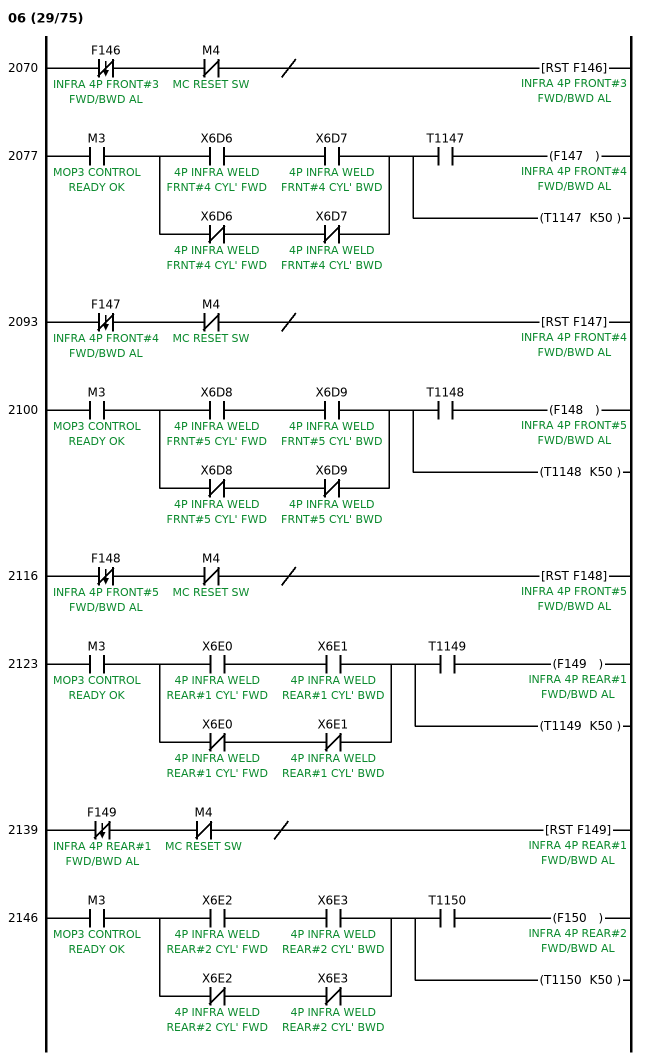
2070  LDFI    F146  ; INFRA 4P FRONT#3 FWD/BWD AL
      ANI     M4  ; MC RESET SW
      INV
      RST     F146  ; INFRA 4P FRONT#3 FWD/BWD AL
2077  LD      M3  ; MOP3 CONTROL READY OK
      LD      X6D6  ; 4P INFRA WELD FRNT#4 CYL' FWD
      AND     X6D7  ; 4P INFRA WELD FRNT#4 CYL' BWD
      LDI     X6D6  ; 4P INFRA WELD FRNT#4 CYL' FWD
      ANI     X6D7  ; 4P INFRA WELD FRNT#4 CYL' BWD
      ORB
      ANB
      MPS
      AND     T1147
      OUT     F147  ; INFRA 4P FRONT#4 FWD/BWD AL
      MPP
      OUT     T1147 K50
2093  LDFI    F147  ; INFRA 4P FRONT#4 FWD/BWD AL
      ANI     M4  ; MC RESET SW
      INV
      RST     F147  ; INFRA 4P FRONT#4 FWD/BWD AL
2100  LD      M3  ; MOP3 CONTROL READY OK
      LD      X6D8  ; 4P INFRA WELD FRNT#5 CYL' FWD
      AND     X6D9  ; 4P INFRA WELD FRNT#5 CYL' BWD
      LDI     X6D8  ; 4P INFRA WELD FRNT#5 CYL' FWD
      ANI     X6D9  ; 4P INFRA WELD FRNT#5 CYL' BWD
      ORB
      ANB
      MPS
      AND     T1148
      OUT     F148  ; INFRA 4P FRONT#5 FWD/BWD AL
      MPP
      OUT     T1148 K50
2116  LDFI    F148  ; INFRA 4P FRONT#5 FWD/BWD AL
      ANI     M4  ; MC RESET SW
      INV
      RST     F148  ; INFRA 4P FRONT#5 FWD/BWD AL
2123  LD      M3  ; MOP3 CONTROL READY OK
      LD      X6E0  ; 4P INFRA WELD REAR#1 CYL' FWD
      AND     X6E1  ; 4P INFRA WELD REAR#1 CYL' BWD
      LDI     X6E0  ; 4P INFRA WELD REAR#1 CYL' FWD
      ANI     X6E1  ; 4P INFRA WELD REAR#1 CYL' BWD
      ORB
      ANB
      MPS
      AND     T1149
      OUT     F149  ; INFRA 4P REAR#1 FWD/BWD AL
      MPP
      OUT     T1149 K50
2139  LDFI    F149  ; INFRA 4P REAR#1 FWD/BWD AL
      ANI     M4  ; MC RESET SW
      INV
      RST     F149  ; INFRA 4P REAR#1 FWD/BWD AL
2146  LD      M3  ; MOP3 CONTROL READY OK
      LD      X6E2  ; 4P INFRA WELD REAR#2 CYL' FWD
      AND     X6E3  ; 4P INFRA WELD REAR#2 CYL' BWD
      LDI     X6E2  ; 4P INFRA WELD REAR#2 CYL' FWD
      ANI     X6E3  ; 4P INFRA WELD REAR#2 CYL' BWD
      ORB
      ANB
      MPS
      AND     T1150
      OUT     F150  ; INFRA 4P REAR#2 FWD/BWD AL
      MPP
      OUT     T1150 K50
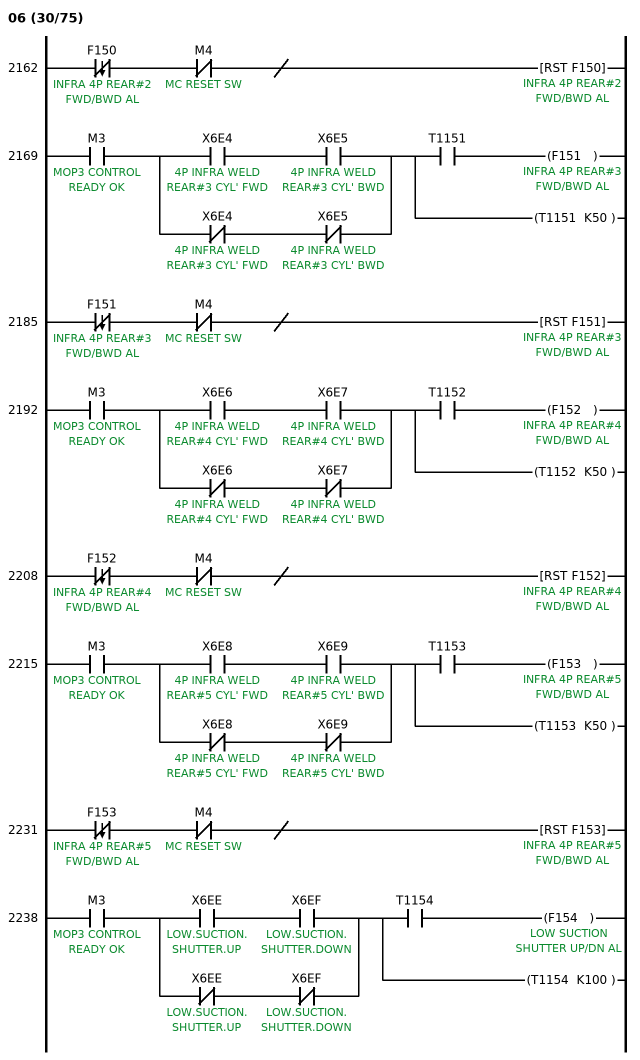
2162  LDFI    F150  ; INFRA 4P REAR#2 FWD/BWD AL
      ANI     M4  ; MC RESET SW
      INV
      RST     F150  ; INFRA 4P REAR#2 FWD/BWD AL
2169  LD      M3  ; MOP3 CONTROL READY OK
      LD      X6E4  ; 4P INFRA WELD REAR#3 CYL' FWD
      AND     X6E5  ; 4P INFRA WELD REAR#3 CYL' BWD
      LDI     X6E4  ; 4P INFRA WELD REAR#3 CYL' FWD
      ANI     X6E5  ; 4P INFRA WELD REAR#3 CYL' BWD
      ORB
      ANB
      MPS
      AND     T1151
      OUT     F151  ; INFRA 4P REAR#3 FWD/BWD AL
      MPP
      OUT     T1151 K50
2185  LDFI    F151  ; INFRA 4P REAR#3 FWD/BWD AL
      ANI     M4  ; MC RESET SW
      INV
      RST     F151  ; INFRA 4P REAR#3 FWD/BWD AL
2192  LD      M3  ; MOP3 CONTROL READY OK
      LD      X6E6  ; 4P INFRA WELD REAR#4 CYL' FWD
      AND     X6E7  ; 4P INFRA WELD REAR#4 CYL' BWD
      LDI     X6E6  ; 4P INFRA WELD REAR#4 CYL' FWD
      ANI     X6E7  ; 4P INFRA WELD REAR#4 CYL' BWD
      ORB
      ANB
      MPS
      AND     T1152
      OUT     F152  ; INFRA 4P REAR#4 FWD/BWD AL
      MPP
      OUT     T1152 K50
2208  LDFI    F152  ; INFRA 4P REAR#4 FWD/BWD AL
      ANI     M4  ; MC RESET SW
      INV
      RST     F152  ; INFRA 4P REAR#4 FWD/BWD AL
2215  LD      M3  ; MOP3 CONTROL READY OK
      LD      X6E8  ; 4P INFRA WELD REAR#5 CYL' FWD
      AND     X6E9  ; 4P INFRA WELD REAR#5 CYL' BWD
      LDI     X6E8  ; 4P INFRA WELD REAR#5 CYL' FWD
      ANI     X6E9  ; 4P INFRA WELD REAR#5 CYL' BWD
      ORB
      ANB
      MPS
      AND     T1153
      OUT     F153  ; INFRA 4P REAR#5 FWD/BWD AL
      MPP
      OUT     T1153 K50
2231  LDFI    F153  ; INFRA 4P REAR#5 FWD/BWD AL
      ANI     M4  ; MC RESET SW
      INV
      RST     F153  ; INFRA 4P REAR#5 FWD/BWD AL
2238  LD      M3  ; MOP3 CONTROL READY OK
      LD      X6EE  ; LOW.SUCTION.SHUTTER.UP
      AND     X6EF  ; LOW.SUCTION.SHUTTER.DOWN
      LDI     X6EE  ; LOW.SUCTION.SHUTTER.UP
      ANI     X6EF  ; LOW.SUCTION.SHUTTER.DOWN
      ORB
      ANB
      MPS
      AND     T1154
      OUT     F154  ; LOW SUCTION SHUTTER UP/DN AL
      MPP
      OUT     T1154 K100
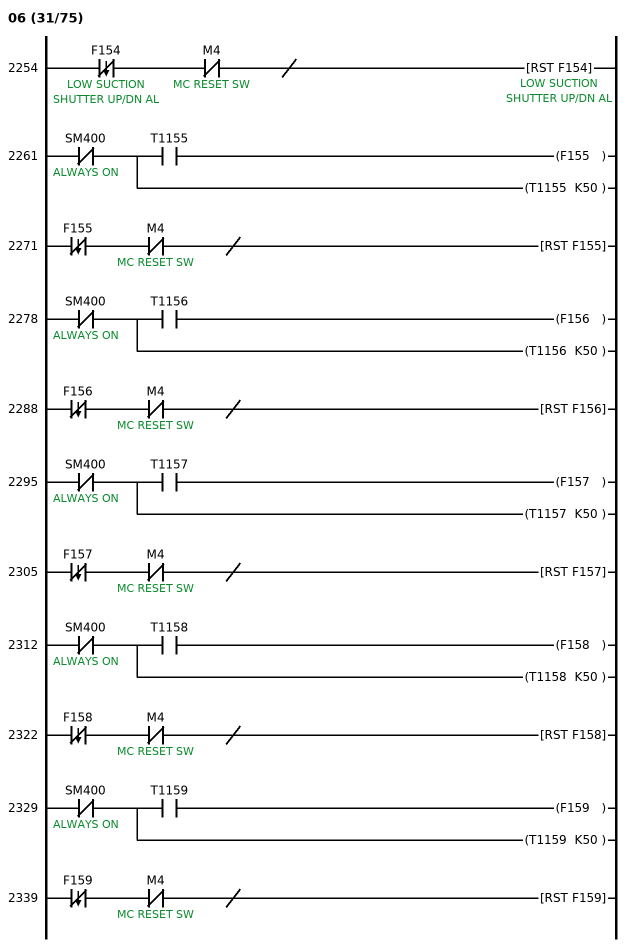
2254  LDFI    F154  ; LOW SUCTION SHUTTER UP/DN AL
      ANI     M4  ; MC RESET SW
      INV
      RST     F154  ; LOW SUCTION SHUTTER UP/DN AL
2261  LDI     SM400  ; ALWAYS ON
      MPS
      AND     T1155
      OUT     F155
      MPP
      OUT     T1155 K50
2271  LDFI    F155
      ANI     M4  ; MC RESET SW
      INV
      RST     F155
2278  LDI     SM400  ; ALWAYS ON
      MPS
      AND     T1156
      OUT     F156
      MPP
      OUT     T1156 K50
2288  LDFI    F156
      ANI     M4  ; MC RESET SW
      INV
      RST     F156
2295  LDI     SM400  ; ALWAYS ON
      MPS
      AND     T1157
      OUT     F157
      MPP
      OUT     T1157 K50
2305  LDFI    F157
      ANI     M4  ; MC RESET SW
      INV
      RST     F157
2312  LDI     SM400  ; ALWAYS ON
      MPS
      AND     T1158
      OUT     F158
      MPP
      OUT     T1158 K50
2322  LDFI    F158
      ANI     M4  ; MC RESET SW
      INV
      RST     F158
2329  LDI     SM400  ; ALWAYS ON
      MPS
      AND     T1159
      OUT     F159
      MPP
      OUT     T1159 K50
2339  LDFI    F159
      ANI     M4  ; MC RESET SW
      INV
      RST     F159
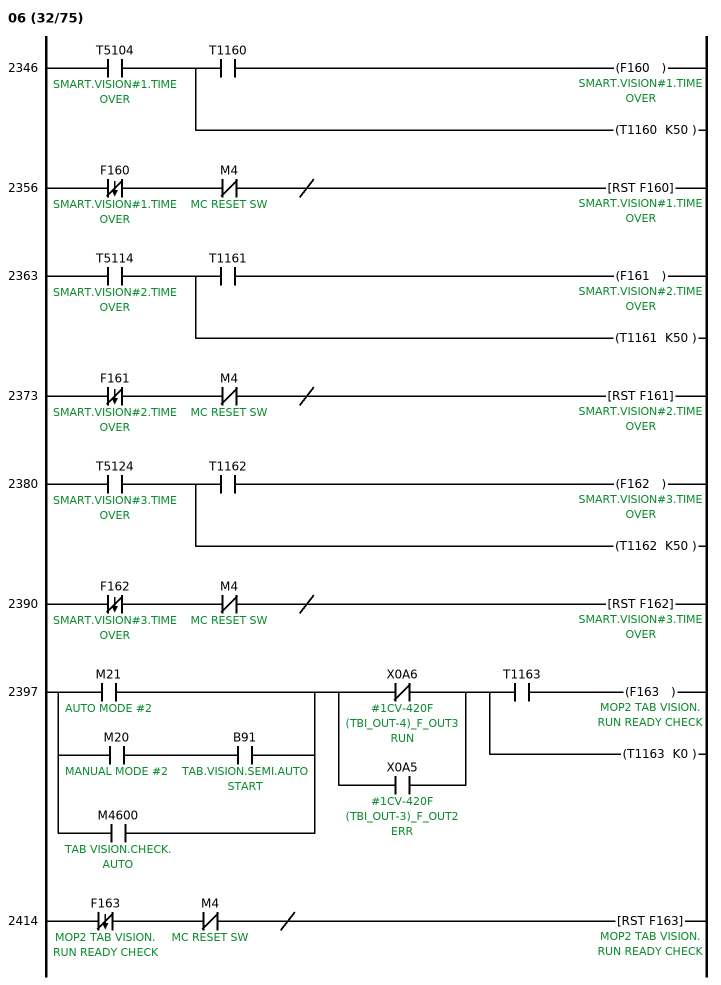
2346  LD      T5104  ; SMART.VISION#1.TIME OVER
      MPS
      AND     T1160
      OUT     F160  ; SMART.VISION#1.TIME OVER
      MPP
      OUT     T1160 K50
2356  LDFI    F160  ; SMART.VISION#1.TIME OVER
      ANI     M4  ; MC RESET SW
      INV
      RST     F160  ; SMART.VISION#1.TIME OVER
2363  LD      T5114  ; SMART.VISION#2.TIME OVER
      MPS
      AND     T1161
      OUT     F161  ; SMART.VISION#2.TIME OVER
      MPP
      OUT     T1161 K50
2373  LDFI    F161  ; SMART.VISION#2.TIME OVER
      ANI     M4  ; MC RESET SW
      INV
      RST     F161  ; SMART.VISION#2.TIME OVER
2380  LD      T5124  ; SMART.VISION#3.TIME OVER
      MPS
      AND     T1162
      OUT     F162  ; SMART.VISION#3.TIME OVER
      MPP
      OUT     T1162 K50
2390  LDFI    F162  ; SMART.VISION#3.TIME OVER
      ANI     M4  ; MC RESET SW
      INV
      RST     F162  ; SMART.VISION#3.TIME OVER
2397  LD      M21  ; AUTO MODE #2
      LD      M20  ; MANUAL MODE #2
      AND     B91  ; TAB.VISION.SEMI.AUTO START
      ORB
      OR      M4600  ; TAB VISION.CHECK.AUTO
      LDI     X0A6  ; #1CV-420F (TBI_OUT-4)_F_OUT3 RUN
      OR      X0A5  ; #1CV-420F (TBI_OUT-3)_F_OUT2 ERR
      ANB
      MPS
      AND     T1163
      OUT     F163  ; MOP2 TAB VISION. RUN READY CHECK
      MPP
      OUT     T1163 K0
2414  LDFI    F163  ; MOP2 TAB VISION. RUN READY CHECK
      ANI     M4  ; MC RESET SW
      INV
      RST     F163  ; MOP2 TAB VISION. RUN READY CHECK
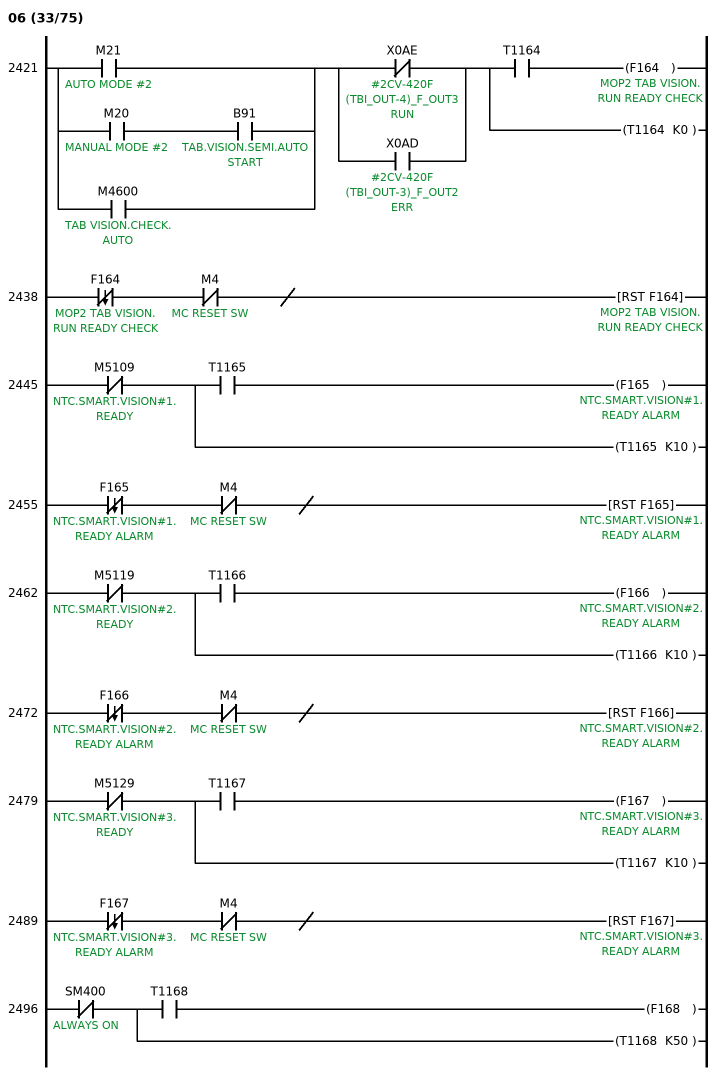
2421  LD      M21  ; AUTO MODE #2
      LD      M20  ; MANUAL MODE #2
      AND     B91  ; TAB.VISION.SEMI.AUTO START
      ORB
      OR      M4600  ; TAB VISION.CHECK.AUTO
      LDI     X0AE  ; #2CV-420F (TBI_OUT-4)_F_OUT3 RUN
      OR      X0AD  ; #2CV-420F (TBI_OUT-3)_F_OUT2 ERR
      ANB
      MPS
      AND     T1164
      OUT     F164  ; MOP2 TAB VISION. RUN READY CHECK
      MPP
      OUT     T1164 K0
2438  LDFI    F164  ; MOP2 TAB VISION. RUN READY CHECK
      ANI     M4  ; MC RESET SW
      INV
      RST     F164  ; MOP2 TAB VISION. RUN READY CHECK
2445  LDI     M5109  ; NTC.SMART.VISION#1.READY
      MPS
      AND     T1165
      OUT     F165  ; NTC.SMART.VISION#1.READY ALARM
      MPP
      OUT     T1165 K10
2455  LDFI    F165  ; NTC.SMART.VISION#1.READY ALARM
      ANI     M4  ; MC RESET SW
      INV
      RST     F165  ; NTC.SMART.VISION#1.READY ALARM
2462  LDI     M5119  ; NTC.SMART.VISION#2.READY
      MPS
      AND     T1166
      OUT     F166  ; NTC.SMART.VISION#2.READY ALARM
      MPP
      OUT     T1166 K10
2472  LDFI    F166  ; NTC.SMART.VISION#2.READY ALARM
      ANI     M4  ; MC RESET SW
      INV
      RST     F166  ; NTC.SMART.VISION#2.READY ALARM
2479  LDI     M5129  ; NTC.SMART.VISION#3.READY
      MPS
      AND     T1167
      OUT     F167  ; NTC.SMART.VISION#3.READY ALARM
      MPP
      OUT     T1167 K10
2489  LDFI    F167  ; NTC.SMART.VISION#3.READY ALARM
      ANI     M4  ; MC RESET SW
      INV
      RST     F167  ; NTC.SMART.VISION#3.READY ALARM
2496  LDI     SM400  ; ALWAYS ON
      MPS
      AND     T1168
      OUT     F168
      MPP
      OUT     T1168 K50
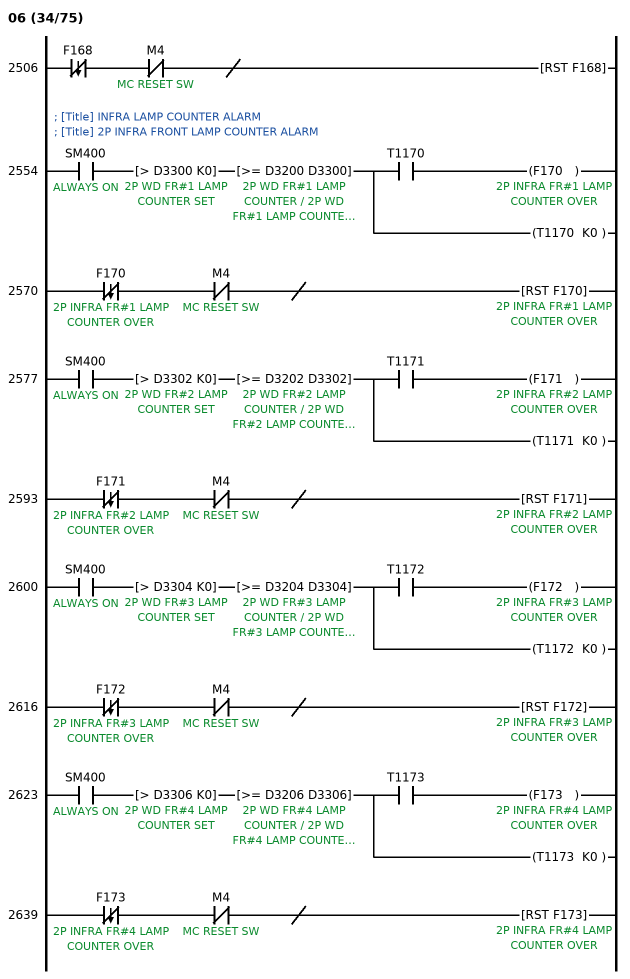
2506  LDFI    F168
      ANI     M4  ; MC RESET SW
      INV
      RST     F168
; [Title] INFRA LAMP COUNTER ALARM
; [Title] 2P INFRA FRONT LAMP COUNTER ALARM
2554  LD      SM400  ; ALWAYS ON
      AND>    D3300 K0  ; 2P WD FR#1 LAMP COUNTER SET
      AND>=   D3200 D3300  ; 2P WD FR#1 LAMP COUNTER / 2P WD FR#1 LAMP COUNTER SET
      MPS
      AND     T1170
      OUT     F170  ; 2P INFRA FR#1 LAMP COUNTER OVER
      MPP
      OUT     T1170 K0
2570  LDFI    F170  ; 2P INFRA FR#1 LAMP COUNTER OVER
      ANI     M4  ; MC RESET SW
      INV
      RST     F170  ; 2P INFRA FR#1 LAMP COUNTER OVER
2577  LD      SM400  ; ALWAYS ON
      AND>    D3302 K0  ; 2P WD FR#2 LAMP COUNTER SET
      AND>=   D3202 D3302  ; 2P WD FR#2 LAMP COUNTER / 2P WD FR#2 LAMP COUNTER SET
      MPS
      AND     T1171
      OUT     F171  ; 2P INFRA FR#2 LAMP COUNTER OVER
      MPP
      OUT     T1171 K0
2593  LDFI    F171  ; 2P INFRA FR#2 LAMP COUNTER OVER
      ANI     M4  ; MC RESET SW
      INV
      RST     F171  ; 2P INFRA FR#2 LAMP COUNTER OVER
2600  LD      SM400  ; ALWAYS ON
      AND>    D3304 K0  ; 2P WD FR#3 LAMP COUNTER SET
      AND>=   D3204 D3304  ; 2P WD FR#3 LAMP COUNTER / 2P WD FR#3 LAMP COUNTER SET
      MPS
      AND     T1172
      OUT     F172  ; 2P INFRA FR#3 LAMP COUNTER OVER
      MPP
      OUT     T1172 K0
2616  LDFI    F172  ; 2P INFRA FR#3 LAMP COUNTER OVER
      ANI     M4  ; MC RESET SW
      INV
      RST     F172  ; 2P INFRA FR#3 LAMP COUNTER OVER
2623  LD      SM400  ; ALWAYS ON
      AND>    D3306 K0  ; 2P WD FR#4 LAMP COUNTER SET
      AND>=   D3206 D3306  ; 2P WD FR#4 LAMP COUNTER / 2P WD FR#4 LAMP COUNTER SET
      MPS
      AND     T1173
      OUT     F173  ; 2P INFRA FR#4 LAMP COUNTER OVER
      MPP
      OUT     T1173 K0
2639  LDFI    F173  ; 2P INFRA FR#4 LAMP COUNTER OVER
      ANI     M4  ; MC RESET SW
      INV
      RST     F173  ; 2P INFRA FR#4 LAMP COUNTER OVER
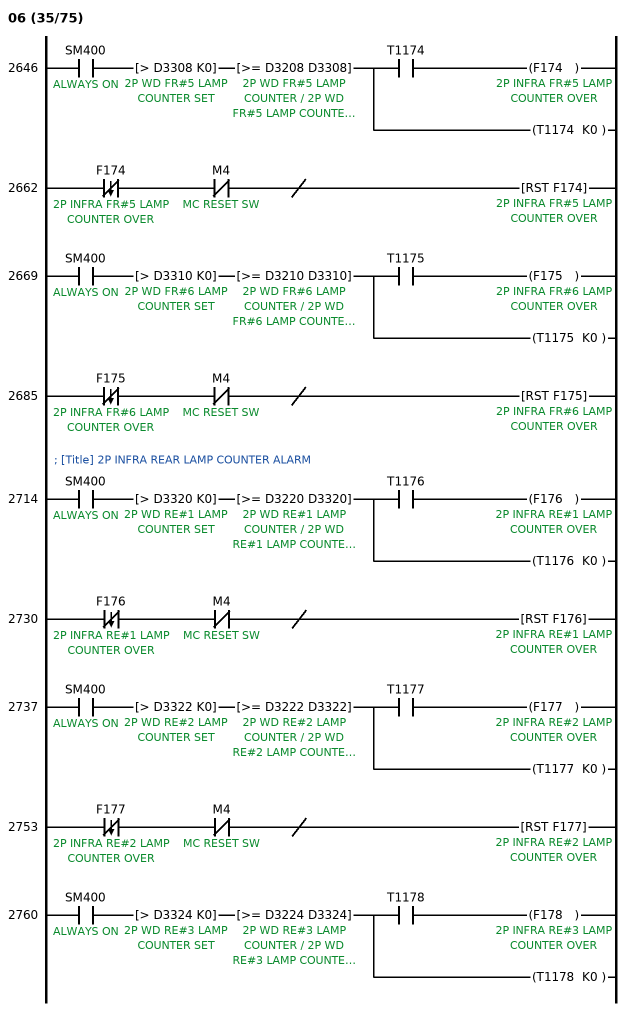
2646  LD      SM400  ; ALWAYS ON
      AND>    D3308 K0  ; 2P WD FR#5 LAMP COUNTER SET
      AND>=   D3208 D3308  ; 2P WD FR#5 LAMP COUNTER / 2P WD FR#5 LAMP COUNTER SET
      MPS
      AND     T1174
      OUT     F174  ; 2P INFRA FR#5 LAMP COUNTER OVER
      MPP
      OUT     T1174 K0
2662  LDFI    F174  ; 2P INFRA FR#5 LAMP COUNTER OVER
      ANI     M4  ; MC RESET SW
      INV
      RST     F174  ; 2P INFRA FR#5 LAMP COUNTER OVER
2669  LD      SM400  ; ALWAYS ON
      AND>    D3310 K0  ; 2P WD FR#6 LAMP COUNTER SET
      AND>=   D3210 D3310  ; 2P WD FR#6 LAMP COUNTER / 2P WD FR#6 LAMP COUNTER SET
      MPS
      AND     T1175
      OUT     F175  ; 2P INFRA FR#6 LAMP COUNTER OVER
      MPP
      OUT     T1175 K0
2685  LDFI    F175  ; 2P INFRA FR#6 LAMP COUNTER OVER
      ANI     M4  ; MC RESET SW
      INV
      RST     F175  ; 2P INFRA FR#6 LAMP COUNTER OVER
; [Title] 2P INFRA REAR LAMP COUNTER ALARM
2714  LD      SM400  ; ALWAYS ON
      AND>    D3320 K0  ; 2P WD RE#1 LAMP COUNTER SET
      AND>=   D3220 D3320  ; 2P WD RE#1 LAMP COUNTER / 2P WD RE#1 LAMP COUNTER SET
      MPS
      AND     T1176
      OUT     F176  ; 2P INFRA RE#1 LAMP COUNTER OVER
      MPP
      OUT     T1176 K0
2730  LDFI    F176  ; 2P INFRA RE#1 LAMP COUNTER OVER
      ANI     M4  ; MC RESET SW
      INV
      RST     F176  ; 2P INFRA RE#1 LAMP COUNTER OVER
2737  LD      SM400  ; ALWAYS ON
      AND>    D3322 K0  ; 2P WD RE#2 LAMP COUNTER SET
      AND>=   D3222 D3322  ; 2P WD RE#2 LAMP COUNTER / 2P WD RE#2 LAMP COUNTER SET
      MPS
      AND     T1177
      OUT     F177  ; 2P INFRA RE#2 LAMP COUNTER OVER
      MPP
      OUT     T1177 K0
2753  LDFI    F177  ; 2P INFRA RE#2 LAMP COUNTER OVER
      ANI     M4  ; MC RESET SW
      INV
      RST     F177  ; 2P INFRA RE#2 LAMP COUNTER OVER
2760  LD      SM400  ; ALWAYS ON
      AND>    D3324 K0  ; 2P WD RE#3 LAMP COUNTER SET
      AND>=   D3224 D3324  ; 2P WD RE#3 LAMP COUNTER / 2P WD RE#3 LAMP COUNTER SET
      MPS
      AND     T1178
      OUT     F178  ; 2P INFRA RE#3 LAMP COUNTER OVER
      MPP
      OUT     T1178 K0
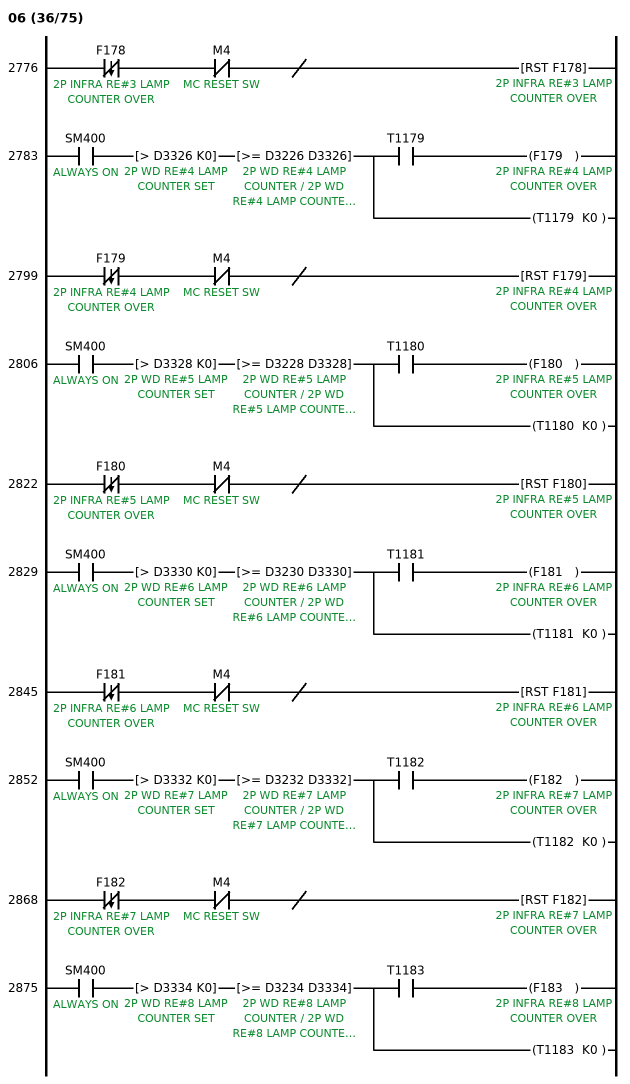
2776  LDFI    F178  ; 2P INFRA RE#3 LAMP COUNTER OVER
      ANI     M4  ; MC RESET SW
      INV
      RST     F178  ; 2P INFRA RE#3 LAMP COUNTER OVER
2783  LD      SM400  ; ALWAYS ON
      AND>    D3326 K0  ; 2P WD RE#4 LAMP COUNTER SET
      AND>=   D3226 D3326  ; 2P WD RE#4 LAMP COUNTER / 2P WD RE#4 LAMP COUNTER SET
      MPS
      AND     T1179
      OUT     F179  ; 2P INFRA RE#4 LAMP COUNTER OVER
      MPP
      OUT     T1179 K0
2799  LDFI    F179  ; 2P INFRA RE#4 LAMP COUNTER OVER
      ANI     M4  ; MC RESET SW
      INV
      RST     F179  ; 2P INFRA RE#4 LAMP COUNTER OVER
2806  LD      SM400  ; ALWAYS ON
      AND>    D3328 K0  ; 2P WD RE#5 LAMP COUNTER SET
      AND>=   D3228 D3328  ; 2P WD RE#5 LAMP COUNTER / 2P WD RE#5 LAMP COUNTER SET
      MPS
      AND     T1180
      OUT     F180  ; 2P INFRA RE#5 LAMP COUNTER OVER
      MPP
      OUT     T1180 K0
2822  LDFI    F180  ; 2P INFRA RE#5 LAMP COUNTER OVER
      ANI     M4  ; MC RESET SW
      INV
      RST     F180  ; 2P INFRA RE#5 LAMP COUNTER OVER
2829  LD      SM400  ; ALWAYS ON
      AND>    D3330 K0  ; 2P WD RE#6 LAMP COUNTER SET
      AND>=   D3230 D3330  ; 2P WD RE#6 LAMP COUNTER / 2P WD RE#6 LAMP COUNTER SET
      MPS
      AND     T1181
      OUT     F181  ; 2P INFRA RE#6 LAMP COUNTER OVER
      MPP
      OUT     T1181 K0
2845  LDFI    F181  ; 2P INFRA RE#6 LAMP COUNTER OVER
      ANI     M4  ; MC RESET SW
      INV
      RST     F181  ; 2P INFRA RE#6 LAMP COUNTER OVER
2852  LD      SM400  ; ALWAYS ON
      AND>    D3332 K0  ; 2P WD RE#7 LAMP COUNTER SET
      AND>=   D3232 D3332  ; 2P WD RE#7 LAMP COUNTER / 2P WD RE#7 LAMP COUNTER SET
      MPS
      AND     T1182
      OUT     F182  ; 2P INFRA RE#7 LAMP COUNTER OVER
      MPP
      OUT     T1182 K0
2868  LDFI    F182  ; 2P INFRA RE#7 LAMP COUNTER OVER
      ANI     M4  ; MC RESET SW
      INV
      RST     F182  ; 2P INFRA RE#7 LAMP COUNTER OVER
2875  LD      SM400  ; ALWAYS ON
      AND>    D3334 K0  ; 2P WD RE#8 LAMP COUNTER SET
      AND>=   D3234 D3334  ; 2P WD RE#8 LAMP COUNTER / 2P WD RE#8 LAMP COUNTER SET
      MPS
      AND     T1183
      OUT     F183  ; 2P INFRA RE#8 LAMP COUNTER OVER
      MPP
      OUT     T1183 K0
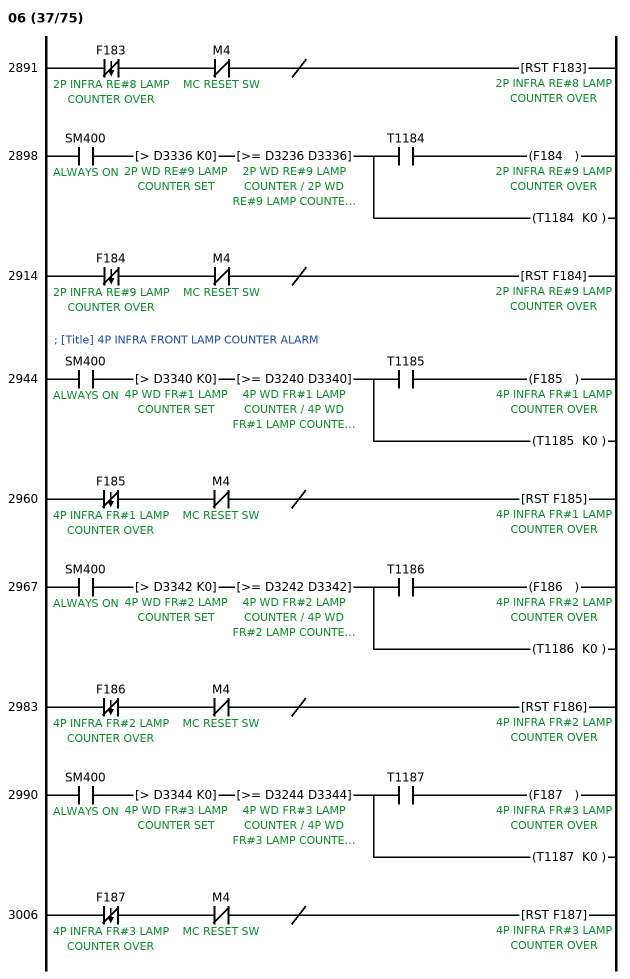
2891  LDFI    F183  ; 2P INFRA RE#8 LAMP COUNTER OVER
      ANI     M4  ; MC RESET SW
      INV
      RST     F183  ; 2P INFRA RE#8 LAMP COUNTER OVER
2898  LD      SM400  ; ALWAYS ON
      AND>    D3336 K0  ; 2P WD RE#9 LAMP COUNTER SET
      AND>=   D3236 D3336  ; 2P WD RE#9 LAMP COUNTER / 2P WD RE#9 LAMP COUNTER SET
      MPS
      AND     T1184
      OUT     F184  ; 2P INFRA RE#9 LAMP COUNTER OVER
      MPP
      OUT     T1184 K0
2914  LDFI    F184  ; 2P INFRA RE#9 LAMP COUNTER OVER
      ANI     M4  ; MC RESET SW
      INV
      RST     F184  ; 2P INFRA RE#9 LAMP COUNTER OVER
; [Title] 4P INFRA FRONT LAMP COUNTER ALARM
2944  LD      SM400  ; ALWAYS ON
      AND>    D3340 K0  ; 4P WD FR#1 LAMP COUNTER SET
      AND>=   D3240 D3340  ; 4P WD FR#1 LAMP COUNTER / 4P WD FR#1 LAMP COUNTER SET
      MPS
      AND     T1185
      OUT     F185  ; 4P INFRA FR#1 LAMP COUNTER OVER
      MPP
      OUT     T1185 K0
2960  LDFI    F185  ; 4P INFRA FR#1 LAMP COUNTER OVER
      ANI     M4  ; MC RESET SW
      INV
      RST     F185  ; 4P INFRA FR#1 LAMP COUNTER OVER
2967  LD      SM400  ; ALWAYS ON
      AND>    D3342 K0  ; 4P WD FR#2 LAMP COUNTER SET
      AND>=   D3242 D3342  ; 4P WD FR#2 LAMP COUNTER / 4P WD FR#2 LAMP COUNTER SET
      MPS
      AND     T1186
      OUT     F186  ; 4P INFRA FR#2 LAMP COUNTER OVER
      MPP
      OUT     T1186 K0
2983  LDFI    F186  ; 4P INFRA FR#2 LAMP COUNTER OVER
      ANI     M4  ; MC RESET SW
      INV
      RST     F186  ; 4P INFRA FR#2 LAMP COUNTER OVER
2990  LD      SM400  ; ALWAYS ON
      AND>    D3344 K0  ; 4P WD FR#3 LAMP COUNTER SET
      AND>=   D3244 D3344  ; 4P WD FR#3 LAMP COUNTER / 4P WD FR#3 LAMP COUNTER SET
      MPS
      AND     T1187
      OUT     F187  ; 4P INFRA FR#3 LAMP COUNTER OVER
      MPP
      OUT     T1187 K0
3006  LDFI    F187  ; 4P INFRA FR#3 LAMP COUNTER OVER
      ANI     M4  ; MC RESET SW
      INV
      RST     F187  ; 4P INFRA FR#3 LAMP COUNTER OVER
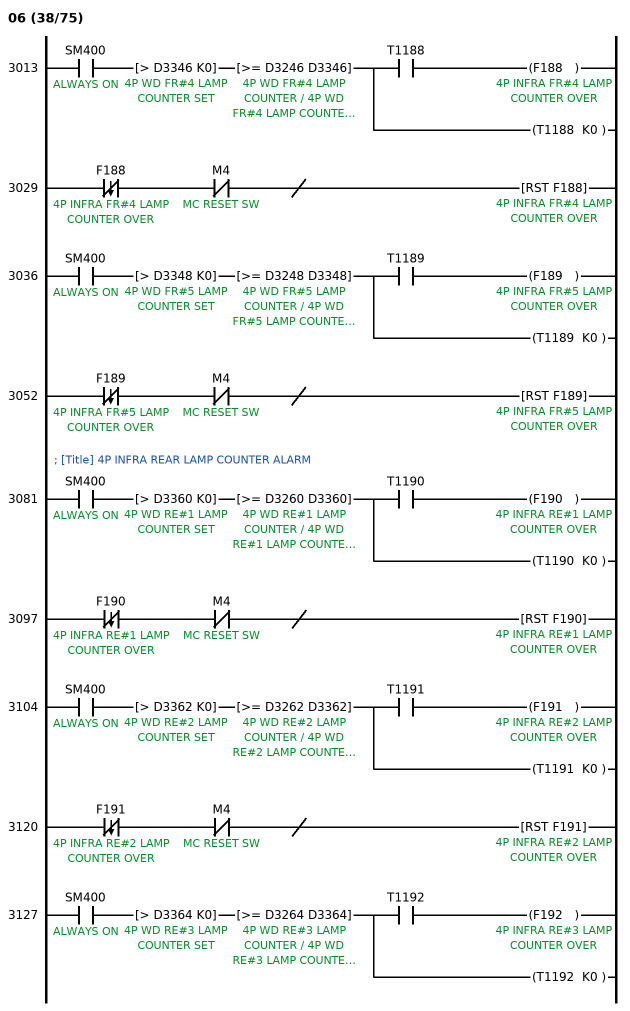
3013  LD      SM400  ; ALWAYS ON
      AND>    D3346 K0  ; 4P WD FR#4 LAMP COUNTER SET
      AND>=   D3246 D3346  ; 4P WD FR#4 LAMP COUNTER / 4P WD FR#4 LAMP COUNTER SET
      MPS
      AND     T1188
      OUT     F188  ; 4P INFRA FR#4 LAMP COUNTER OVER
      MPP
      OUT     T1188 K0
3029  LDFI    F188  ; 4P INFRA FR#4 LAMP COUNTER OVER
      ANI     M4  ; MC RESET SW
      INV
      RST     F188  ; 4P INFRA FR#4 LAMP COUNTER OVER
3036  LD      SM400  ; ALWAYS ON
      AND>    D3348 K0  ; 4P WD FR#5 LAMP COUNTER SET
      AND>=   D3248 D3348  ; 4P WD FR#5 LAMP COUNTER / 4P WD FR#5 LAMP COUNTER SET
      MPS
      AND     T1189
      OUT     F189  ; 4P INFRA FR#5 LAMP COUNTER OVER
      MPP
      OUT     T1189 K0
3052  LDFI    F189  ; 4P INFRA FR#5 LAMP COUNTER OVER
      ANI     M4  ; MC RESET SW
      INV
      RST     F189  ; 4P INFRA FR#5 LAMP COUNTER OVER
; [Title] 4P INFRA REAR LAMP COUNTER ALARM
3081  LD      SM400  ; ALWAYS ON
      AND>    D3360 K0  ; 4P WD RE#1 LAMP COUNTER SET
      AND>=   D3260 D3360  ; 4P WD RE#1 LAMP COUNTER / 4P WD RE#1 LAMP COUNTER SET
      MPS
      AND     T1190
      OUT     F190  ; 4P INFRA RE#1 LAMP COUNTER OVER
      MPP
      OUT     T1190 K0
3097  LDFI    F190  ; 4P INFRA RE#1 LAMP COUNTER OVER
      ANI     M4  ; MC RESET SW
      INV
      RST     F190  ; 4P INFRA RE#1 LAMP COUNTER OVER
3104  LD      SM400  ; ALWAYS ON
      AND>    D3362 K0  ; 4P WD RE#2 LAMP COUNTER SET
      AND>=   D3262 D3362  ; 4P WD RE#2 LAMP COUNTER / 4P WD RE#2 LAMP COUNTER SET
      MPS
      AND     T1191
      OUT     F191  ; 4P INFRA RE#2 LAMP COUNTER OVER
      MPP
      OUT     T1191 K0
3120  LDFI    F191  ; 4P INFRA RE#2 LAMP COUNTER OVER
      ANI     M4  ; MC RESET SW
      INV
      RST     F191  ; 4P INFRA RE#2 LAMP COUNTER OVER
3127  LD      SM400  ; ALWAYS ON
      AND>    D3364 K0  ; 4P WD RE#3 LAMP COUNTER SET
      AND>=   D3264 D3364  ; 4P WD RE#3 LAMP COUNTER / 4P WD RE#3 LAMP COUNTER SET
      MPS
      AND     T1192
      OUT     F192  ; 4P INFRA RE#3 LAMP COUNTER OVER
      MPP
      OUT     T1192 K0
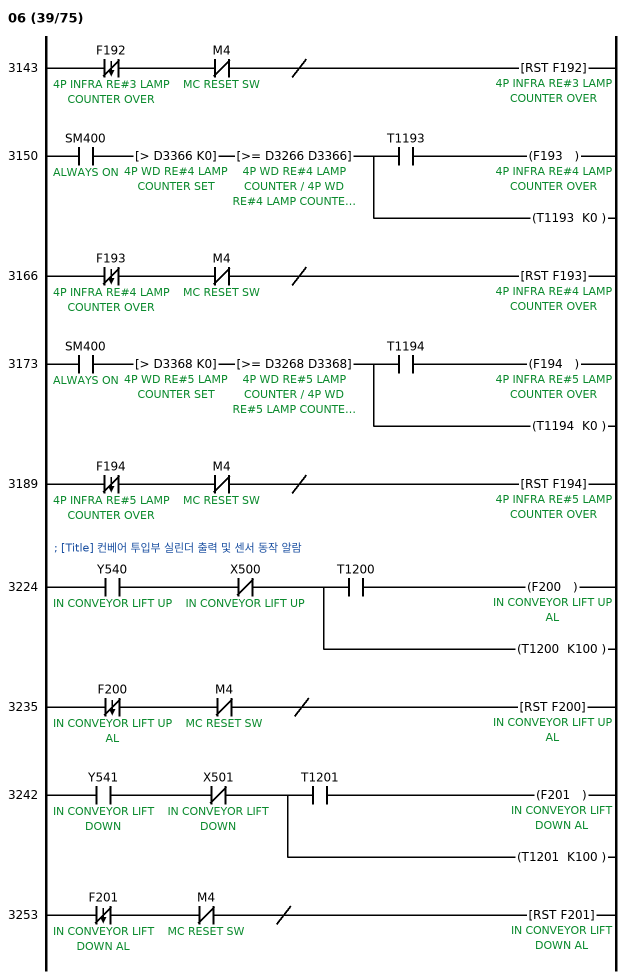
3143  LDFI    F192  ; 4P INFRA RE#3 LAMP COUNTER OVER
      ANI     M4  ; MC RESET SW
      INV
      RST     F192  ; 4P INFRA RE#3 LAMP COUNTER OVER
3150  LD      SM400  ; ALWAYS ON
      AND>    D3366 K0  ; 4P WD RE#4 LAMP COUNTER SET
      AND>=   D3266 D3366  ; 4P WD RE#4 LAMP COUNTER / 4P WD RE#4 LAMP COUNTER SET
      MPS
      AND     T1193
      OUT     F193  ; 4P INFRA RE#4 LAMP COUNTER OVER
      MPP
      OUT     T1193 K0
3166  LDFI    F193  ; 4P INFRA RE#4 LAMP COUNTER OVER
      ANI     M4  ; MC RESET SW
      INV
      RST     F193  ; 4P INFRA RE#4 LAMP COUNTER OVER
3173  LD      SM400  ; ALWAYS ON
      AND>    D3368 K0  ; 4P WD RE#5 LAMP COUNTER SET
      AND>=   D3268 D3368  ; 4P WD RE#5 LAMP COUNTER / 4P WD RE#5 LAMP COUNTER SET
      MPS
      AND     T1194
      OUT     F194  ; 4P INFRA RE#5 LAMP COUNTER OVER
      MPP
      OUT     T1194 K0
3189  LDFI    F194  ; 4P INFRA RE#5 LAMP COUNTER OVER
      ANI     M4  ; MC RESET SW
      INV
      RST     F194  ; 4P INFRA RE#5 LAMP COUNTER OVER
; [Title] 컨베어 투입부 실린더 출력 및 센서 동작 알람
3224  LD      Y540  ; IN CONVEYOR LIFT UP
      ANI     X500  ; IN CONVEYOR LIFT UP
      MPS
      AND     T1200
      OUT     F200  ; IN CONVEYOR LIFT UP AL
      MPP
      OUT     T1200 K100
3235  LDFI    F200  ; IN CONVEYOR LIFT UP AL
      ANI     M4  ; MC RESET SW
      INV
      RST     F200  ; IN CONVEYOR LIFT UP AL
3242  LD      Y541  ; IN CONVEYOR LIFT DOWN
      ANI     X501  ; IN CONVEYOR LIFT DOWN
      MPS
      AND     T1201
      OUT     F201  ; IN CONVEYOR LIFT DOWN AL
      MPP
      OUT     T1201 K100
3253  LDFI    F201  ; IN CONVEYOR LIFT DOWN AL
      ANI     M4  ; MC RESET SW
      INV
      RST     F201  ; IN CONVEYOR LIFT DOWN AL
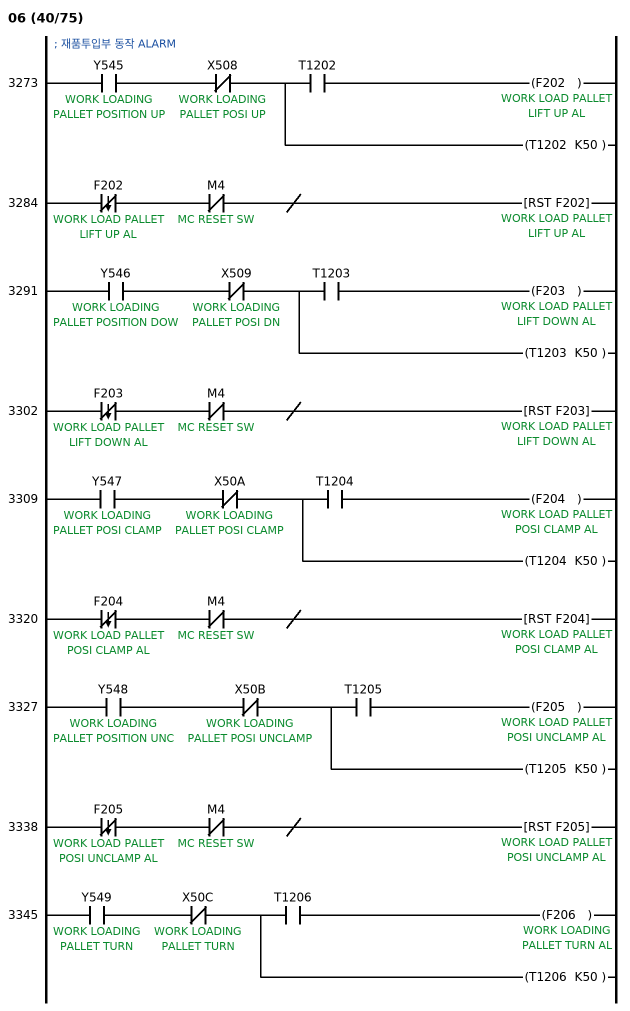
; 재품투입부 동작 ALARM
3273  LD      Y545  ; WORK LOADING PALLET POSITION UP
      ANI     X508  ; WORK LOADING PALLET POSI UP
      MPS
      AND     T1202
      OUT     F202  ; WORK LOAD PALLET LIFT UP AL
      MPP
      OUT     T1202 K50
3284  LDFI    F202  ; WORK LOAD PALLET LIFT UP AL
      ANI     M4  ; MC RESET SW
      INV
      RST     F202  ; WORK LOAD PALLET LIFT UP AL
3291  LD      Y546  ; WORK LOADING PALLET POSITION DOW
      ANI     X509  ; WORK LOADING PALLET POSI DN
      MPS
      AND     T1203
      OUT     F203  ; WORK LOAD PALLET LIFT DOWN AL
      MPP
      OUT     T1203 K50
3302  LDFI    F203  ; WORK LOAD PALLET LIFT DOWN AL
      ANI     M4  ; MC RESET SW
      INV
      RST     F203  ; WORK LOAD PALLET LIFT DOWN AL
3309  LD      Y547  ; WORK LOADING PALLET POSI CLAMP
      ANI     X50A  ; WORK LOADING PALLET POSI CLAMP
      MPS
      AND     T1204
      OUT     F204  ; WORK LOAD PALLET POSI CLAMP AL
      MPP
      OUT     T1204 K50
3320  LDFI    F204  ; WORK LOAD PALLET POSI CLAMP AL
      ANI     M4  ; MC RESET SW
      INV
      RST     F204  ; WORK LOAD PALLET POSI CLAMP AL
3327  LD      Y548  ; WORK LOADING PALLET POSITION UNC
      ANI     X50B  ; WORK LOADING PALLET POSI UNCLAMP
      MPS
      AND     T1205
      OUT     F205  ; WORK LOAD PALLET POSI UNCLAMP AL
      MPP
      OUT     T1205 K50
3338  LDFI    F205  ; WORK LOAD PALLET POSI UNCLAMP AL
      ANI     M4  ; MC RESET SW
      INV
      RST     F205  ; WORK LOAD PALLET POSI UNCLAMP AL
3345  LD      Y549  ; WORK LOADING PALLET TURN
      ANI     X50C  ; WORK LOADING PALLET TURN
      MPS
      AND     T1206
      OUT     F206  ; WORK LOADING PALLET TURN AL
      MPP
      OUT     T1206 K50
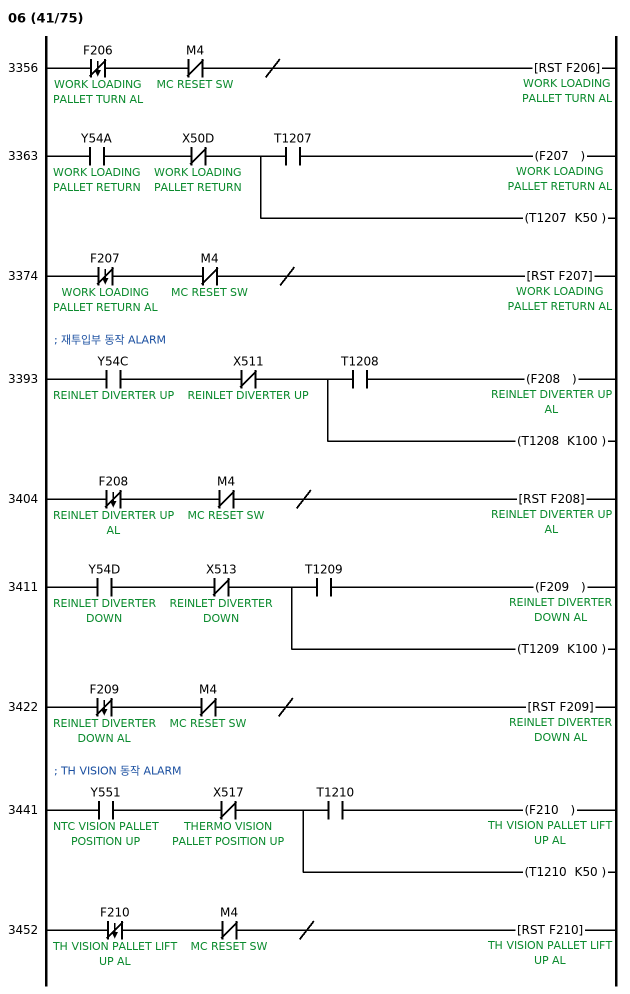
3356  LDFI    F206  ; WORK LOADING PALLET TURN AL
      ANI     M4  ; MC RESET SW
      INV
      RST     F206  ; WORK LOADING PALLET TURN AL
3363  LD      Y54A  ; WORK LOADING PALLET RETURN
      ANI     X50D  ; WORK LOADING PALLET RETURN
      MPS
      AND     T1207
      OUT     F207  ; WORK LOADING PALLET RETURN AL
      MPP
      OUT     T1207 K50
3374  LDFI    F207  ; WORK LOADING PALLET RETURN AL
      ANI     M4  ; MC RESET SW
      INV
      RST     F207  ; WORK LOADING PALLET RETURN AL
; 재투입부 동작 ALARM
3393  LD      Y54C  ; REINLET DIVERTER UP
      ANI     X511  ; REINLET DIVERTER UP
      MPS
      AND     T1208
      OUT     F208  ; REINLET DIVERTER UP AL
      MPP
      OUT     T1208 K100
3404  LDFI    F208  ; REINLET DIVERTER UP AL
      ANI     M4  ; MC RESET SW
      INV
      RST     F208  ; REINLET DIVERTER UP AL
3411  LD      Y54D  ; REINLET DIVERTER DOWN
      ANI     X513  ; REINLET DIVERTER DOWN
      MPS
      AND     T1209
      OUT     F209  ; REINLET DIVERTER DOWN AL
      MPP
      OUT     T1209 K100
3422  LDFI    F209  ; REINLET DIVERTER DOWN AL
      ANI     M4  ; MC RESET SW
      INV
      RST     F209  ; REINLET DIVERTER DOWN AL
; TH VISION 동작 ALARM
3441  LD      Y551  ; NTC VISION PALLET POSITION UP
      ANI     X517  ; THERMO VISION PALLET POSITION UP
      MPS
      AND     T1210
      OUT     F210  ; TH VISION PALLET LIFT UP AL
      MPP
      OUT     T1210 K50
3452  LDFI    F210  ; TH VISION PALLET LIFT UP AL
      ANI     M4  ; MC RESET SW
      INV
      RST     F210  ; TH VISION PALLET LIFT UP AL
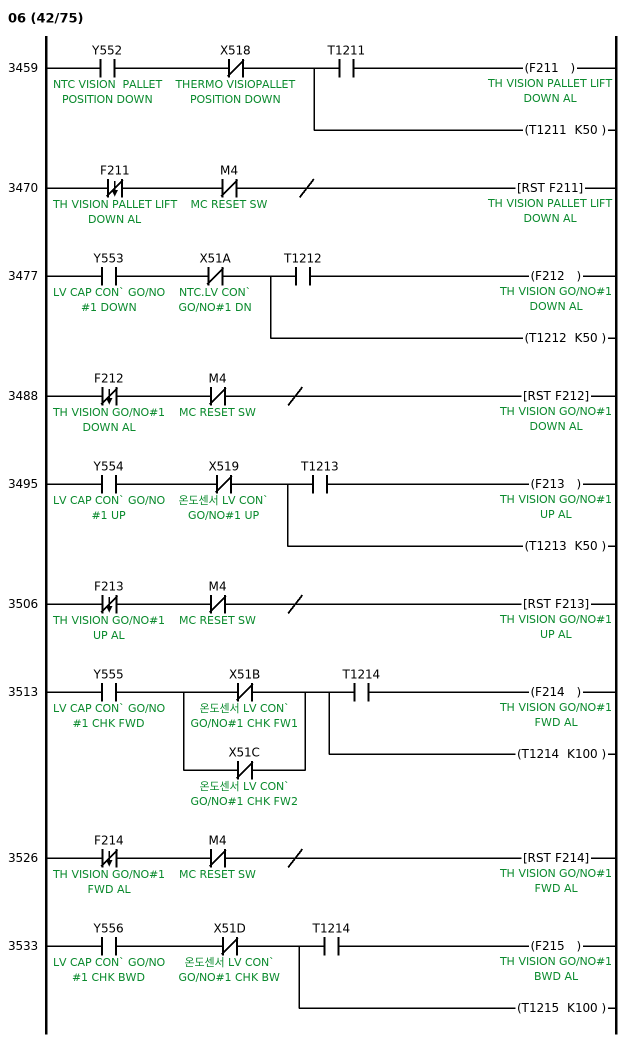
3459  LD      Y552  ; NTC VISION  PALLET POSITION DOWN
      ANI     X518  ; THERMO VISIOPALLET POSITION DOWN
      MPS
      AND     T1211
      OUT     F211  ; TH VISION PALLET LIFT DOWN AL
      MPP
      OUT     T1211 K50
3470  LDFI    F211  ; TH VISION PALLET LIFT DOWN AL
      ANI     M4  ; MC RESET SW
      INV
      RST     F211  ; TH VISION PALLET LIFT DOWN AL
3477  LD      Y553  ; LV CAP CON` GO/NO #1 DOWN
      ANI     X51A  ; NTC.LV CON` GO/NO#1 DN
      MPS
      AND     T1212
      OUT     F212  ; TH VISION GO/NO#1 DOWN AL
      MPP
      OUT     T1212 K50
3488  LDFI    F212  ; TH VISION GO/NO#1 DOWN AL
      ANI     M4  ; MC RESET SW
      INV
      RST     F212  ; TH VISION GO/NO#1 DOWN AL
3495  LD      Y554  ; LV CAP CON` GO/NO #1 UP
      ANI     X519  ; 온도센서 LV CON` GO/NO#1 UP
      MPS
      AND     T1213
      OUT     F213  ; TH VISION GO/NO#1 UP AL
      MPP
      OUT     T1213 K50
3506  LDFI    F213  ; TH VISION GO/NO#1 UP AL
      ANI     M4  ; MC RESET SW
      INV
      RST     F213  ; TH VISION GO/NO#1 UP AL
3513  LD      Y555  ; LV CAP CON` GO/NO #1 CHK FWD
      LDI     X51B  ; 온도센서 LV CON` GO/NO#1 CHK FW1
      ORI     X51C  ; 온도센서 LV CON` GO/NO#1 CHK FW2
      ANB
      MPS
      AND     T1214
      OUT     F214  ; TH VISION GO/NO#1 FWD AL
      MPP
      OUT     T1214 K100
3526  LDFI    F214  ; TH VISION GO/NO#1 FWD AL
      ANI     M4  ; MC RESET SW
      INV
      RST     F214  ; TH VISION GO/NO#1 FWD AL
3533  LD      Y556  ; LV CAP CON` GO/NO #1 CHK BWD
      ANI     X51D  ; 온도센서 LV CON` GO/NO#1 CHK BW
      MPS
      AND     T1214
      OUT     F215  ; TH VISION GO/NO#1 BWD AL
      MPP
      OUT     T1215 K100
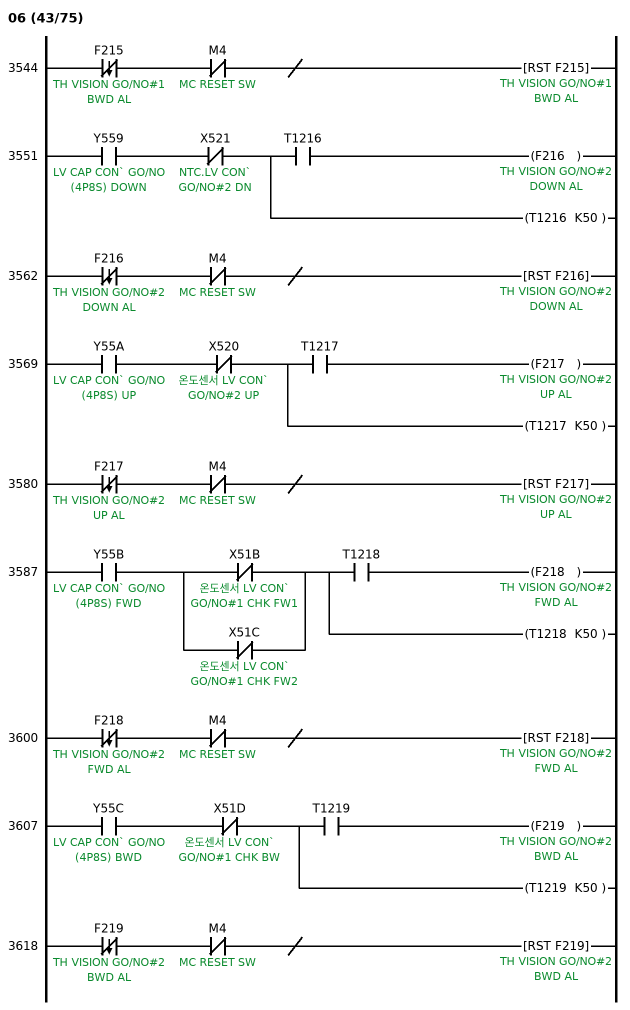
3544  LDFI    F215  ; TH VISION GO/NO#1 BWD AL
      ANI     M4  ; MC RESET SW
      INV
      RST     F215  ; TH VISION GO/NO#1 BWD AL
3551  LD      Y559  ; LV CAP CON` GO/NO (4P8S) DOWN
      ANI     X521  ; NTC.LV CON` GO/NO#2 DN
      MPS
      AND     T1216
      OUT     F216  ; TH VISION GO/NO#2 DOWN AL
      MPP
      OUT     T1216 K50
3562  LDFI    F216  ; TH VISION GO/NO#2 DOWN AL
      ANI     M4  ; MC RESET SW
      INV
      RST     F216  ; TH VISION GO/NO#2 DOWN AL
3569  LD      Y55A  ; LV CAP CON` GO/NO (4P8S) UP
      ANI     X520  ; 온도센서 LV CON` GO/NO#2 UP
      MPS
      AND     T1217
      OUT     F217  ; TH VISION GO/NO#2 UP AL
      MPP
      OUT     T1217 K50
3580  LDFI    F217  ; TH VISION GO/NO#2 UP AL
      ANI     M4  ; MC RESET SW
      INV
      RST     F217  ; TH VISION GO/NO#2 UP AL
3587  LD      Y55B  ; LV CAP CON` GO/NO (4P8S) FWD
      LDI     X51B  ; 온도센서 LV CON` GO/NO#1 CHK FW1
      ORI     X51C  ; 온도센서 LV CON` GO/NO#1 CHK FW2
      ANB
      MPS
      AND     T1218
      OUT     F218  ; TH VISION GO/NO#2 FWD AL
      MPP
      OUT     T1218 K50
3600  LDFI    F218  ; TH VISION GO/NO#2 FWD AL
      ANI     M4  ; MC RESET SW
      INV
      RST     F218  ; TH VISION GO/NO#2 FWD AL
3607  LD      Y55C  ; LV CAP CON` GO/NO (4P8S) BWD
      ANI     X51D  ; 온도센서 LV CON` GO/NO#1 CHK BW
      MPS
      AND     T1219
      OUT     F219  ; TH VISION GO/NO#2 BWD AL
      MPP
      OUT     T1219 K50
3618  LDFI    F219  ; TH VISION GO/NO#2 BWD AL
      ANI     M4  ; MC RESET SW
      INV
      RST     F219  ; TH VISION GO/NO#2 BWD AL
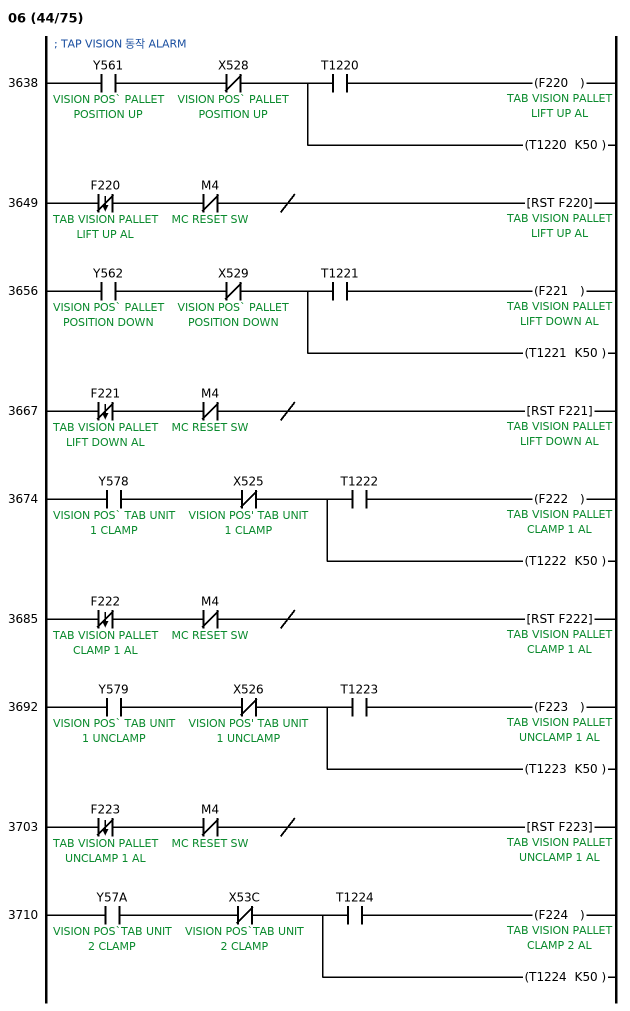
; TAP VISION 동작 ALARM
3638  LD      Y561  ; VISION POS` PALLET POSITION UP
      ANI     X528  ; VISION POS` PALLET POSITION UP
      MPS
      AND     T1220
      OUT     F220  ; TAB VISION PALLET LIFT UP AL
      MPP
      OUT     T1220 K50
3649  LDFI    F220  ; TAB VISION PALLET LIFT UP AL
      ANI     M4  ; MC RESET SW
      INV
      RST     F220  ; TAB VISION PALLET LIFT UP AL
3656  LD      Y562  ; VISION POS` PALLET POSITION DOWN
      ANI     X529  ; VISION POS` PALLET POSITION DOWN
      MPS
      AND     T1221
      OUT     F221  ; TAB VISION PALLET LIFT DOWN AL
      MPP
      OUT     T1221 K50
3667  LDFI    F221  ; TAB VISION PALLET LIFT DOWN AL
      ANI     M4  ; MC RESET SW
      INV
      RST     F221  ; TAB VISION PALLET LIFT DOWN AL
3674  LD      Y578  ; VISION POS` TAB UNIT 1 CLAMP
      ANI     X525  ; VISION POS' TAB UNIT 1 CLAMP
      MPS
      AND     T1222
      OUT     F222  ; TAB VISION PALLET CLAMP 1 AL
      MPP
      OUT     T1222 K50
3685  LDFI    F222  ; TAB VISION PALLET CLAMP 1 AL
      ANI     M4  ; MC RESET SW
      INV
      RST     F222  ; TAB VISION PALLET CLAMP 1 AL
3692  LD      Y579  ; VISION POS` TAB UNIT 1 UNCLAMP
      ANI     X526  ; VISION POS' TAB UNIT 1 UNCLAMP
      MPS
      AND     T1223
      OUT     F223  ; TAB VISION PALLET UNCLAMP 1 AL
      MPP
      OUT     T1223 K50
3703  LDFI    F223  ; TAB VISION PALLET UNCLAMP 1 AL
      ANI     M4  ; MC RESET SW
      INV
      RST     F223  ; TAB VISION PALLET UNCLAMP 1 AL
3710  LD      Y57A  ; VISION POS`TAB UNIT 2 CLAMP
      ANI     X53C  ; VISION POS`TAB UNIT 2 CLAMP
      MPS
      AND     T1224
      OUT     F224  ; TAB VISION PALLET CLAMP 2 AL
      MPP
      OUT     T1224 K50
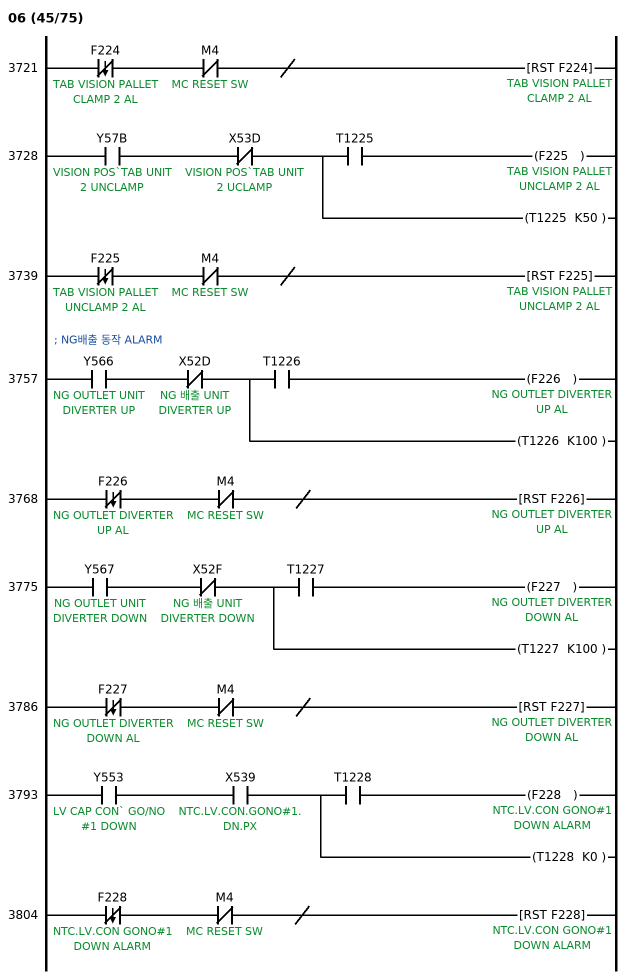
3721  LDFI    F224  ; TAB VISION PALLET CLAMP 2 AL
      ANI     M4  ; MC RESET SW
      INV
      RST     F224  ; TAB VISION PALLET CLAMP 2 AL
3728  LD      Y57B  ; VISION POS`TAB UNIT 2 UNCLAMP
      ANI     X53D  ; VISION POS`TAB UNIT 2 UCLAMP
      MPS
      AND     T1225
      OUT     F225  ; TAB VISION PALLET UNCLAMP 2 AL
      MPP
      OUT     T1225 K50
3739  LDFI    F225  ; TAB VISION PALLET UNCLAMP 2 AL
      ANI     M4  ; MC RESET SW
      INV
      RST     F225  ; TAB VISION PALLET UNCLAMP 2 AL
; NG배출 동작 ALARM
3757  LD      Y566  ; NG OUTLET UNIT DIVERTER UP
      ANI     X52D  ; NG 배출 UNIT DIVERTER UP
      MPS
      AND     T1226
      OUT     F226  ; NG OUTLET DIVERTER UP AL
      MPP
      OUT     T1226 K100
3768  LDFI    F226  ; NG OUTLET DIVERTER UP AL
      ANI     M4  ; MC RESET SW
      INV
      RST     F226  ; NG OUTLET DIVERTER UP AL
3775  LD      Y567  ; NG OUTLET UNIT DIVERTER DOWN
      ANI     X52F  ; NG 배출 UNIT DIVERTER DOWN
      MPS
      AND     T1227
      OUT     F227  ; NG OUTLET DIVERTER DOWN AL
      MPP
      OUT     T1227 K100
3786  LDFI    F227  ; NG OUTLET DIVERTER DOWN AL
      ANI     M4  ; MC RESET SW
      INV
      RST     F227  ; NG OUTLET DIVERTER DOWN AL
3793  LD      Y553  ; LV CAP CON` GO/NO #1 DOWN
      AND     X539  ; NTC.LV.CON.GONO#1.DN.PX
      MPS
      AND     T1228
      OUT     F228  ; NTC.LV.CON GONO#1 DOWN ALARM
      MPP
      OUT     T1228 K0
3804  LDFI    F228  ; NTC.LV.CON GONO#1 DOWN ALARM
      ANI     M4  ; MC RESET SW
      INV
      RST     F228  ; NTC.LV.CON GONO#1 DOWN ALARM
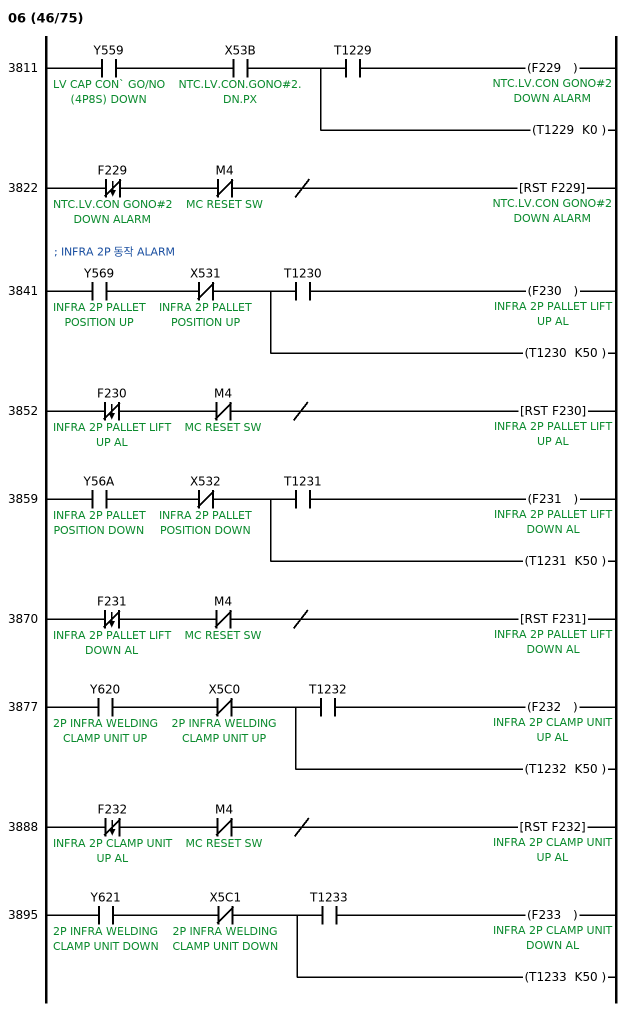
3811  LD      Y559  ; LV CAP CON` GO/NO (4P8S) DOWN
      AND     X53B  ; NTC.LV.CON.GONO#2.DN.PX
      MPS
      AND     T1229
      OUT     F229  ; NTC.LV.CON GONO#2 DOWN ALARM
      MPP
      OUT     T1229 K0
3822  LDFI    F229  ; NTC.LV.CON GONO#2 DOWN ALARM
      ANI     M4  ; MC RESET SW
      INV
      RST     F229  ; NTC.LV.CON GONO#2 DOWN ALARM
; INFRA 2P 동작 ALARM
3841  LD      Y569  ; INFRA 2P PALLET POSITION UP
      ANI     X531  ; INFRA 2P PALLET POSITION UP
      MPS
      AND     T1230
      OUT     F230  ; INFRA 2P PALLET LIFT UP AL
      MPP
      OUT     T1230 K50
3852  LDFI    F230  ; INFRA 2P PALLET LIFT UP AL
      ANI     M4  ; MC RESET SW
      INV
      RST     F230  ; INFRA 2P PALLET LIFT UP AL
3859  LD      Y56A  ; INFRA 2P PALLET POSITION DOWN
      ANI     X532  ; INFRA 2P PALLET POSITION DOWN
      MPS
      AND     T1231
      OUT     F231  ; INFRA 2P PALLET LIFT DOWN AL
      MPP
      OUT     T1231 K50
3870  LDFI    F231  ; INFRA 2P PALLET LIFT DOWN AL
      ANI     M4  ; MC RESET SW
      INV
      RST     F231  ; INFRA 2P PALLET LIFT DOWN AL
3877  LD      Y620  ; 2P INFRA WELDING CLAMP UNIT UP
      ANI     X5C0  ; 2P INFRA WELDING CLAMP UNIT UP
      MPS
      AND     T1232
      OUT     F232  ; INFRA 2P CLAMP UNIT UP AL
      MPP
      OUT     T1232 K50
3888  LDFI    F232  ; INFRA 2P CLAMP UNIT UP AL
      ANI     M4  ; MC RESET SW
      INV
      RST     F232  ; INFRA 2P CLAMP UNIT UP AL
3895  LD      Y621  ; 2P INFRA WELDING CLAMP UNIT DOWN
      ANI     X5C1  ; 2P INFRA WELDING CLAMP UNIT DOWN
      MPS
      AND     T1233
      OUT     F233  ; INFRA 2P CLAMP UNIT DOWN AL
      MPP
      OUT     T1233 K50
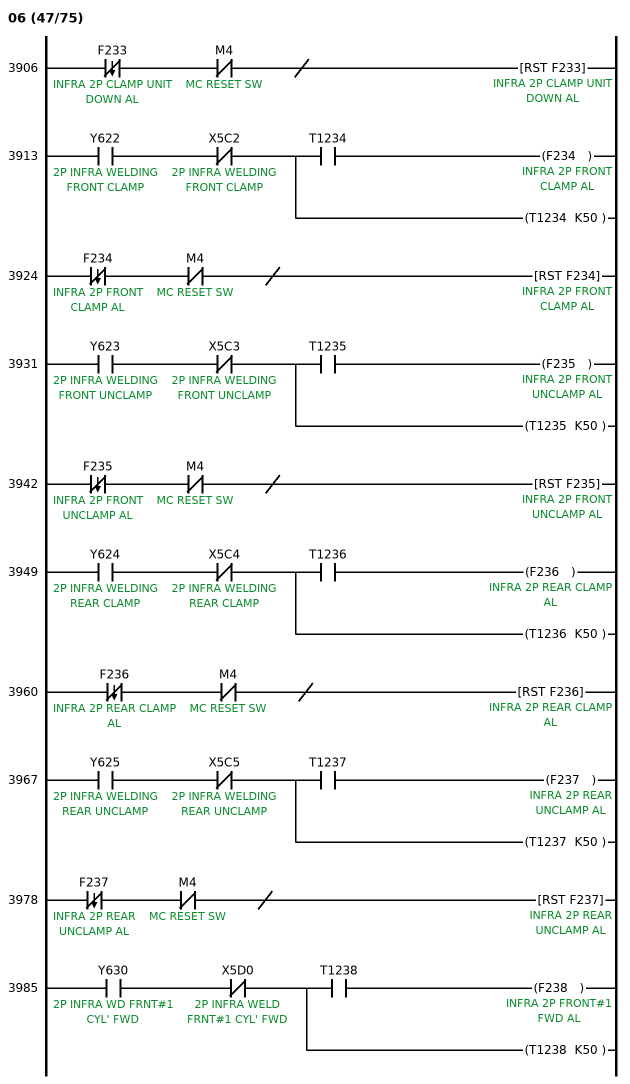
3906  LDFI    F233  ; INFRA 2P CLAMP UNIT DOWN AL
      ANI     M4  ; MC RESET SW
      INV
      RST     F233  ; INFRA 2P CLAMP UNIT DOWN AL
3913  LD      Y622  ; 2P INFRA WELDING FRONT CLAMP
      ANI     X5C2  ; 2P INFRA WELDING FRONT CLAMP
      MPS
      AND     T1234
      OUT     F234  ; INFRA 2P FRONT CLAMP AL
      MPP
      OUT     T1234 K50
3924  LDFI    F234  ; INFRA 2P FRONT CLAMP AL
      ANI     M4  ; MC RESET SW
      INV
      RST     F234  ; INFRA 2P FRONT CLAMP AL
3931  LD      Y623  ; 2P INFRA WELDING FRONT UNCLAMP
      ANI     X5C3  ; 2P INFRA WELDING FRONT UNCLAMP
      MPS
      AND     T1235
      OUT     F235  ; INFRA 2P FRONT UNCLAMP AL
      MPP
      OUT     T1235 K50
3942  LDFI    F235  ; INFRA 2P FRONT UNCLAMP AL
      ANI     M4  ; MC RESET SW
      INV
      RST     F235  ; INFRA 2P FRONT UNCLAMP AL
3949  LD      Y624  ; 2P INFRA WELDING REAR CLAMP
      ANI     X5C4  ; 2P INFRA WELDING REAR CLAMP
      MPS
      AND     T1236
      OUT     F236  ; INFRA 2P REAR CLAMP AL
      MPP
      OUT     T1236 K50
3960  LDFI    F236  ; INFRA 2P REAR CLAMP AL
      ANI     M4  ; MC RESET SW
      INV
      RST     F236  ; INFRA 2P REAR CLAMP AL
3967  LD      Y625  ; 2P INFRA WELDING REAR UNCLAMP
      ANI     X5C5  ; 2P INFRA WELDING REAR UNCLAMP
      MPS
      AND     T1237
      OUT     F237  ; INFRA 2P REAR UNCLAMP AL
      MPP
      OUT     T1237 K50
3978  LDFI    F237  ; INFRA 2P REAR UNCLAMP AL
      ANI     M4  ; MC RESET SW
      INV
      RST     F237  ; INFRA 2P REAR UNCLAMP AL
3985  LD      Y630  ; 2P INFRA WD FRNT#1 CYL' FWD
      ANI     X5D0  ; 2P INFRA WELD FRNT#1 CYL' FWD
      MPS
      AND     T1238
      OUT     F238  ; INFRA 2P FRONT#1 FWD AL
      MPP
      OUT     T1238 K50
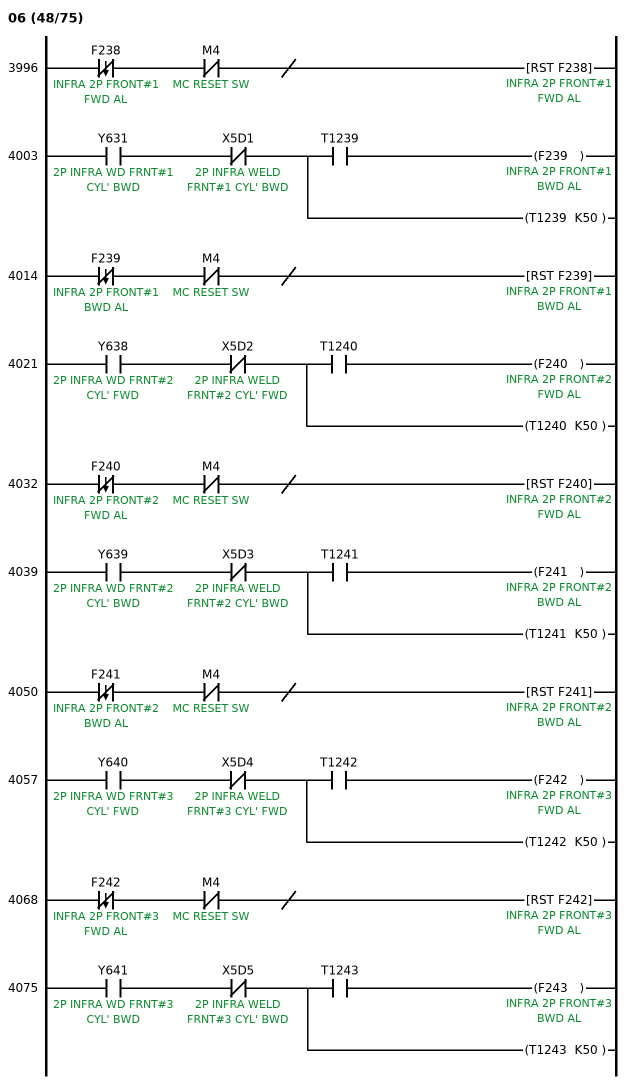
3996  LDFI    F238  ; INFRA 2P FRONT#1 FWD AL
      ANI     M4  ; MC RESET SW
      INV
      RST     F238  ; INFRA 2P FRONT#1 FWD AL
4003  LD      Y631  ; 2P INFRA WD FRNT#1 CYL' BWD
      ANI     X5D1  ; 2P INFRA WELD FRNT#1 CYL' BWD
      MPS
      AND     T1239
      OUT     F239  ; INFRA 2P FRONT#1 BWD AL
      MPP
      OUT     T1239 K50
4014  LDFI    F239  ; INFRA 2P FRONT#1 BWD AL
      ANI     M4  ; MC RESET SW
      INV
      RST     F239  ; INFRA 2P FRONT#1 BWD AL
4021  LD      Y638  ; 2P INFRA WD FRNT#2 CYL' FWD
      ANI     X5D2  ; 2P INFRA WELD FRNT#2 CYL' FWD
      MPS
      AND     T1240
      OUT     F240  ; INFRA 2P FRONT#2 FWD AL
      MPP
      OUT     T1240 K50
4032  LDFI    F240  ; INFRA 2P FRONT#2 FWD AL
      ANI     M4  ; MC RESET SW
      INV
      RST     F240  ; INFRA 2P FRONT#2 FWD AL
4039  LD      Y639  ; 2P INFRA WD FRNT#2 CYL' BWD
      ANI     X5D3  ; 2P INFRA WELD FRNT#2 CYL' BWD
      MPS
      AND     T1241
      OUT     F241  ; INFRA 2P FRONT#2 BWD AL
      MPP
      OUT     T1241 K50
4050  LDFI    F241  ; INFRA 2P FRONT#2 BWD AL
      ANI     M4  ; MC RESET SW
      INV
      RST     F241  ; INFRA 2P FRONT#2 BWD AL
4057  LD      Y640  ; 2P INFRA WD FRNT#3 CYL' FWD
      ANI     X5D4  ; 2P INFRA WELD FRNT#3 CYL' FWD
      MPS
      AND     T1242
      OUT     F242  ; INFRA 2P FRONT#3 FWD AL
      MPP
      OUT     T1242 K50
4068  LDFI    F242  ; INFRA 2P FRONT#3 FWD AL
      ANI     M4  ; MC RESET SW
      INV
      RST     F242  ; INFRA 2P FRONT#3 FWD AL
4075  LD      Y641  ; 2P INFRA WD FRNT#3 CYL' BWD
      ANI     X5D5  ; 2P INFRA WELD FRNT#3 CYL' BWD
      MPS
      AND     T1243
      OUT     F243  ; INFRA 2P FRONT#3 BWD AL
      MPP
      OUT     T1243 K50
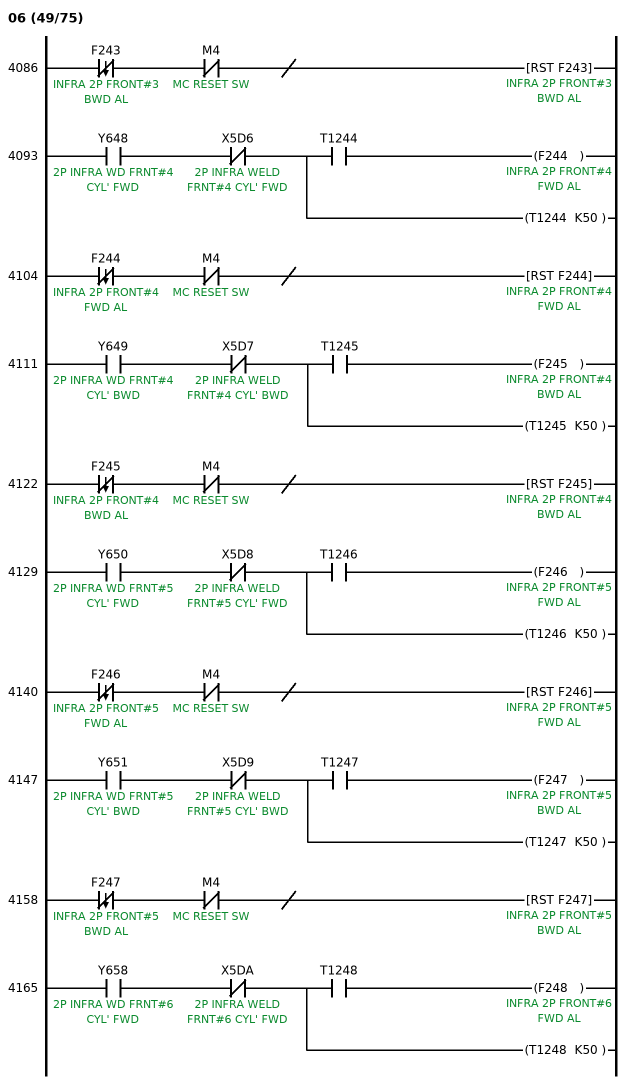
4086  LDFI    F243  ; INFRA 2P FRONT#3 BWD AL
      ANI     M4  ; MC RESET SW
      INV
      RST     F243  ; INFRA 2P FRONT#3 BWD AL
4093  LD      Y648  ; 2P INFRA WD FRNT#4 CYL' FWD
      ANI     X5D6  ; 2P INFRA WELD FRNT#4 CYL' FWD
      MPS
      AND     T1244
      OUT     F244  ; INFRA 2P FRONT#4 FWD AL
      MPP
      OUT     T1244 K50
4104  LDFI    F244  ; INFRA 2P FRONT#4 FWD AL
      ANI     M4  ; MC RESET SW
      INV
      RST     F244  ; INFRA 2P FRONT#4 FWD AL
4111  LD      Y649  ; 2P INFRA WD FRNT#4 CYL' BWD
      ANI     X5D7  ; 2P INFRA WELD FRNT#4 CYL' BWD
      MPS
      AND     T1245
      OUT     F245  ; INFRA 2P FRONT#4 BWD AL
      MPP
      OUT     T1245 K50
4122  LDFI    F245  ; INFRA 2P FRONT#4 BWD AL
      ANI     M4  ; MC RESET SW
      INV
      RST     F245  ; INFRA 2P FRONT#4 BWD AL
4129  LD      Y650  ; 2P INFRA WD FRNT#5 CYL' FWD
      ANI     X5D8  ; 2P INFRA WELD FRNT#5 CYL' FWD
      MPS
      AND     T1246
      OUT     F246  ; INFRA 2P FRONT#5 FWD AL
      MPP
      OUT     T1246 K50
4140  LDFI    F246  ; INFRA 2P FRONT#5 FWD AL
      ANI     M4  ; MC RESET SW
      INV
      RST     F246  ; INFRA 2P FRONT#5 FWD AL
4147  LD      Y651  ; 2P INFRA WD FRNT#5 CYL' BWD
      ANI     X5D9  ; 2P INFRA WELD FRNT#5 CYL' BWD
      MPS
      AND     T1247
      OUT     F247  ; INFRA 2P FRONT#5 BWD AL
      MPP
      OUT     T1247 K50
4158  LDFI    F247  ; INFRA 2P FRONT#5 BWD AL
      ANI     M4  ; MC RESET SW
      INV
      RST     F247  ; INFRA 2P FRONT#5 BWD AL
4165  LD      Y658  ; 2P INFRA WD FRNT#6 CYL' FWD
      ANI     X5DA  ; 2P INFRA WELD FRNT#6 CYL' FWD
      MPS
      AND     T1248
      OUT     F248  ; INFRA 2P FRONT#6 FWD AL
      MPP
      OUT     T1248 K50
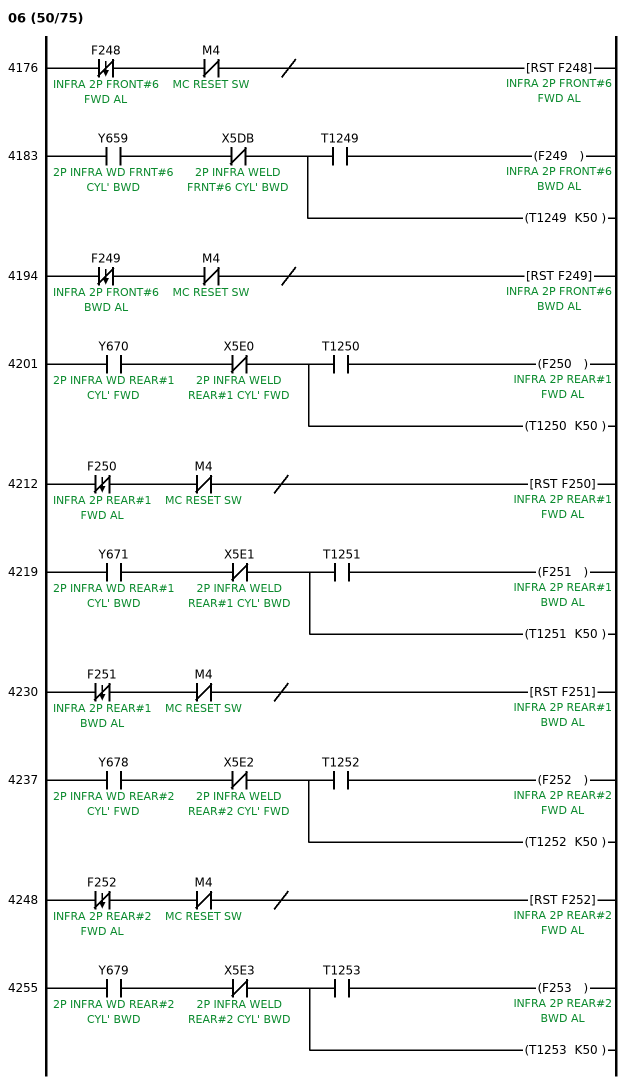
4176  LDFI    F248  ; INFRA 2P FRONT#6 FWD AL
      ANI     M4  ; MC RESET SW
      INV
      RST     F248  ; INFRA 2P FRONT#6 FWD AL
4183  LD      Y659  ; 2P INFRA WD FRNT#6 CYL' BWD
      ANI     X5DB  ; 2P INFRA WELD FRNT#6 CYL' BWD
      MPS
      AND     T1249
      OUT     F249  ; INFRA 2P FRONT#6 BWD AL
      MPP
      OUT     T1249 K50
4194  LDFI    F249  ; INFRA 2P FRONT#6 BWD AL
      ANI     M4  ; MC RESET SW
      INV
      RST     F249  ; INFRA 2P FRONT#6 BWD AL
4201  LD      Y670  ; 2P INFRA WD REAR#1 CYL' FWD
      ANI     X5E0  ; 2P INFRA WELD REAR#1 CYL' FWD
      MPS
      AND     T1250
      OUT     F250  ; INFRA 2P REAR#1 FWD AL
      MPP
      OUT     T1250 K50
4212  LDFI    F250  ; INFRA 2P REAR#1 FWD AL
      ANI     M4  ; MC RESET SW
      INV
      RST     F250  ; INFRA 2P REAR#1 FWD AL
4219  LD      Y671  ; 2P INFRA WD REAR#1 CYL' BWD
      ANI     X5E1  ; 2P INFRA WELD REAR#1 CYL' BWD
      MPS
      AND     T1251
      OUT     F251  ; INFRA 2P REAR#1 BWD AL
      MPP
      OUT     T1251 K50
4230  LDFI    F251  ; INFRA 2P REAR#1 BWD AL
      ANI     M4  ; MC RESET SW
      INV
      RST     F251  ; INFRA 2P REAR#1 BWD AL
4237  LD      Y678  ; 2P INFRA WD REAR#2 CYL' FWD
      ANI     X5E2  ; 2P INFRA WELD REAR#2 CYL' FWD
      MPS
      AND     T1252
      OUT     F252  ; INFRA 2P REAR#2 FWD AL
      MPP
      OUT     T1252 K50
4248  LDFI    F252  ; INFRA 2P REAR#2 FWD AL
      ANI     M4  ; MC RESET SW
      INV
      RST     F252  ; INFRA 2P REAR#2 FWD AL
4255  LD      Y679  ; 2P INFRA WD REAR#2 CYL' BWD
      ANI     X5E3  ; 2P INFRA WELD REAR#2 CYL' BWD
      MPS
      AND     T1253
      OUT     F253  ; INFRA 2P REAR#2 BWD AL
      MPP
      OUT     T1253 K50
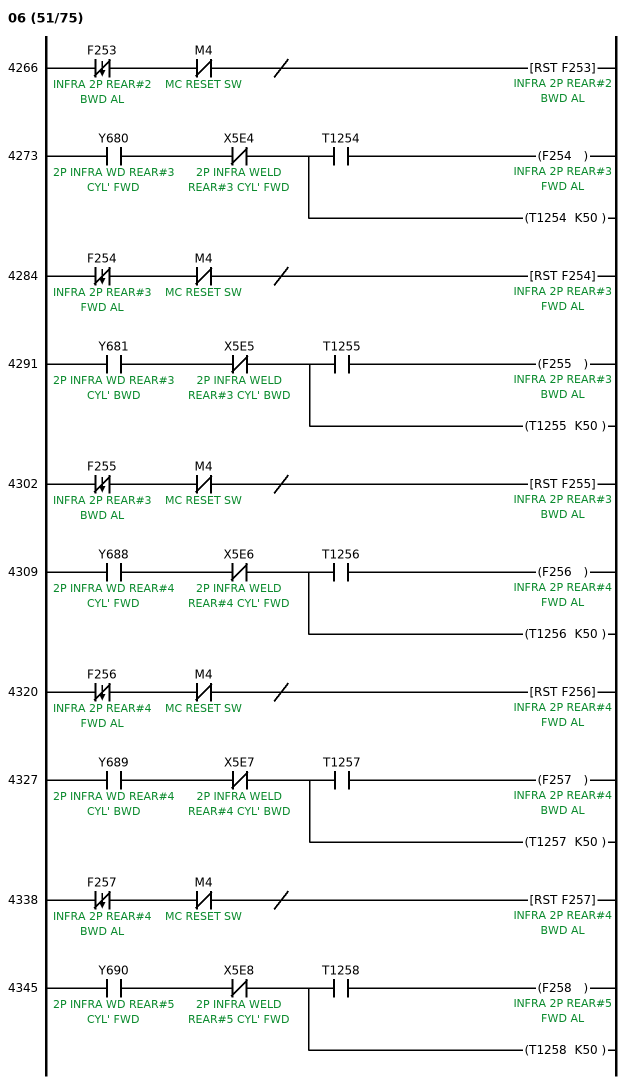
4266  LDFI    F253  ; INFRA 2P REAR#2 BWD AL
      ANI     M4  ; MC RESET SW
      INV
      RST     F253  ; INFRA 2P REAR#2 BWD AL
4273  LD      Y680  ; 2P INFRA WD REAR#3 CYL' FWD
      ANI     X5E4  ; 2P INFRA WELD REAR#3 CYL' FWD
      MPS
      AND     T1254
      OUT     F254  ; INFRA 2P REAR#3 FWD AL
      MPP
      OUT     T1254 K50
4284  LDFI    F254  ; INFRA 2P REAR#3 FWD AL
      ANI     M4  ; MC RESET SW
      INV
      RST     F254  ; INFRA 2P REAR#3 FWD AL
4291  LD      Y681  ; 2P INFRA WD REAR#3 CYL' BWD
      ANI     X5E5  ; 2P INFRA WELD REAR#3 CYL' BWD
      MPS
      AND     T1255
      OUT     F255  ; INFRA 2P REAR#3 BWD AL
      MPP
      OUT     T1255 K50
4302  LDFI    F255  ; INFRA 2P REAR#3 BWD AL
      ANI     M4  ; MC RESET SW
      INV
      RST     F255  ; INFRA 2P REAR#3 BWD AL
4309  LD      Y688  ; 2P INFRA WD REAR#4 CYL' FWD
      ANI     X5E6  ; 2P INFRA WELD REAR#4 CYL' FWD
      MPS
      AND     T1256
      OUT     F256  ; INFRA 2P REAR#4 FWD AL
      MPP
      OUT     T1256 K50
4320  LDFI    F256  ; INFRA 2P REAR#4 FWD AL
      ANI     M4  ; MC RESET SW
      INV
      RST     F256  ; INFRA 2P REAR#4 FWD AL
4327  LD      Y689  ; 2P INFRA WD REAR#4 CYL' BWD
      ANI     X5E7  ; 2P INFRA WELD REAR#4 CYL' BWD
      MPS
      AND     T1257
      OUT     F257  ; INFRA 2P REAR#4 BWD AL
      MPP
      OUT     T1257 K50
4338  LDFI    F257  ; INFRA 2P REAR#4 BWD AL
      ANI     M4  ; MC RESET SW
      INV
      RST     F257  ; INFRA 2P REAR#4 BWD AL
4345  LD      Y690  ; 2P INFRA WD REAR#5 CYL' FWD
      ANI     X5E8  ; 2P INFRA WELD REAR#5 CYL' FWD
      MPS
      AND     T1258
      OUT     F258  ; INFRA 2P REAR#5 FWD AL
      MPP
      OUT     T1258 K50
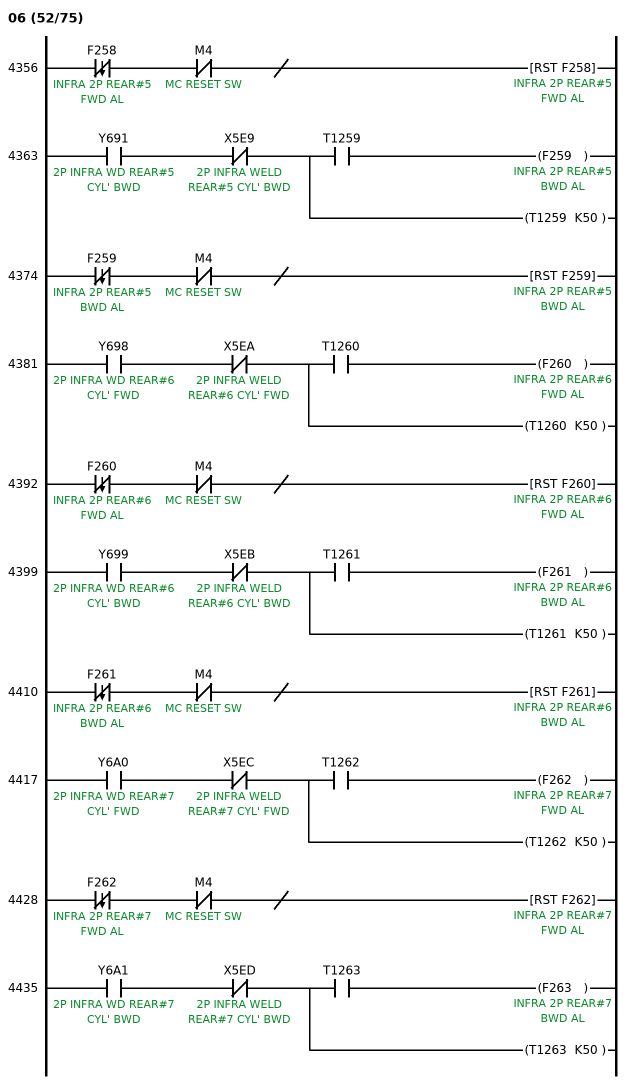
4356  LDFI    F258  ; INFRA 2P REAR#5 FWD AL
      ANI     M4  ; MC RESET SW
      INV
      RST     F258  ; INFRA 2P REAR#5 FWD AL
4363  LD      Y691  ; 2P INFRA WD REAR#5 CYL' BWD
      ANI     X5E9  ; 2P INFRA WELD REAR#5 CYL' BWD
      MPS
      AND     T1259
      OUT     F259  ; INFRA 2P REAR#5 BWD AL
      MPP
      OUT     T1259 K50
4374  LDFI    F259  ; INFRA 2P REAR#5 BWD AL
      ANI     M4  ; MC RESET SW
      INV
      RST     F259  ; INFRA 2P REAR#5 BWD AL
4381  LD      Y698  ; 2P INFRA WD REAR#6 CYL' FWD
      ANI     X5EA  ; 2P INFRA WELD REAR#6 CYL' FWD
      MPS
      AND     T1260
      OUT     F260  ; INFRA 2P REAR#6 FWD AL
      MPP
      OUT     T1260 K50
4392  LDFI    F260  ; INFRA 2P REAR#6 FWD AL
      ANI     M4  ; MC RESET SW
      INV
      RST     F260  ; INFRA 2P REAR#6 FWD AL
4399  LD      Y699  ; 2P INFRA WD REAR#6 CYL' BWD
      ANI     X5EB  ; 2P INFRA WELD REAR#6 CYL' BWD
      MPS
      AND     T1261
      OUT     F261  ; INFRA 2P REAR#6 BWD AL
      MPP
      OUT     T1261 K50
4410  LDFI    F261  ; INFRA 2P REAR#6 BWD AL
      ANI     M4  ; MC RESET SW
      INV
      RST     F261  ; INFRA 2P REAR#6 BWD AL
4417  LD      Y6A0  ; 2P INFRA WD REAR#7 CYL' FWD
      ANI     X5EC  ; 2P INFRA WELD REAR#7 CYL' FWD
      MPS
      AND     T1262
      OUT     F262  ; INFRA 2P REAR#7 FWD AL
      MPP
      OUT     T1262 K50
4428  LDFI    F262  ; INFRA 2P REAR#7 FWD AL
      ANI     M4  ; MC RESET SW
      INV
      RST     F262  ; INFRA 2P REAR#7 FWD AL
4435  LD      Y6A1  ; 2P INFRA WD REAR#7 CYL' BWD
      ANI     X5ED  ; 2P INFRA WELD REAR#7 CYL' BWD
      MPS
      AND     T1263
      OUT     F263  ; INFRA 2P REAR#7 BWD AL
      MPP
      OUT     T1263 K50
